LIN {X 0,Y 298.452,Z 269.609,A -85,B 0,C 180,E1 -16435.587,E2 -16435.587} C_VEL
LIN {X 0,Y 298.198,Z 272.62,A -85,B 0,C 180,E1 -16438.768,E2 -16438.768} C_VEL
LIN {X 0,Y 297.924,Z 275.64,A -85,B 0,C 180,E1 -16441.849,E2 -16441.849} C_VEL
LIN {X 0,Y 297.634,Z 279.334,A -85,B 0,C 180,E1 -16445.446,E2 -16445.446} C_VEL
LIN {X 0,Y 302.181,Z 294.942,A -85,B 0,C 180,E1 -16446.632,E2 -16446.632} C_VEL
LIN {X 0,Y 304.72,Z 306.185,A -85,B 0,C 180,E1 -16447.658,E2 -16447.658} C_VEL
LIN {X 0,Y 306.557,Z 317.092,A -85,B 0,C 180,E1 -16448.834,E2 -16448.834} C_VEL
LIN {X 0,Y 305.846,Z 324.673,A -85,B 0,C 180,E1 -16449.662,E2 -16449.662} C_VEL
LIN {X 0,Y 304.462,Z 334.817,A -85,B 0,C 180,E1 -16450.971,E2 -16450.971} C_VEL
LIN {X 0,Y 303.067,Z 344.133,A -85,B 0,C 180,E1 -16452.454,E2 -16452.454} C_VEL
LIN {X 0,Y 301.645,Z 352.621,A -85,B 0,C 180,E1 -16454.112,E2 -16454.112} C_VEL
LIN {X 0,Y 300.146,Z 360.872,A -85,B 0,C 180,E1 -16456.113,E2 -16456.113} C_VEL
LIN {X 0,Y 299.11,Z 366.515,A -85,B 0,C 180,E1 -16457.792,E2 -16457.792} C_VEL
LIN {X 0,Y 298.156,Z 372.013,A -85,B 0,C 180,E1 -16459.817,E2 -16459.817} C_VEL
LIN {X 0,Y 297.455,Z 376.327,A -85,B 0,C 180,E1 -16461.85,E2 -16461.85} C_VEL
LIN {X 0,Y 297.118,Z 378.98,A -85,B 0,C 180,E1 -16463.448,E2 -16463.448} C_VEL
LIN {X 0,Y 296.782,Z 381.858,A -85,B 0,C 180,E1 -16465.926,E2 -16465.926} C_VEL
LIN {X 0,Y 296.535,Z 383.463,A -85,B 0,C 180,E1 -16468.642,E2 -16468.642} C_VEL
LIN {X 0,Y 296.526,Z 383.693,A -85,B 0,C 180,E1 -16470,E2 -16470} C_VEL
LIN {X 0,Y 296.535,Z 383.502,A -85,B 0,C 180,E1 -16471.358,E2 -16471.358} C_VEL
LIN {X 0,Y 296.779,Z 381.947,A -85,B 0,C 180,E1 -16474.074,E2 -16474.074} C_VEL
LIN {X 0,Y 297.086,Z 379.22,A -85,B 0,C 180,E1 -16476.498,E2 -16476.498} C_VEL
LIN {X 0,Y 297.658,Z 375.251,A -85,B 0,C 180,E1 -16478.828,E2 -16478.828} C_VEL
LIN {X 0,Y 298.411,Z 370.618,A -85,B 0,C 180,E1 -16480.86,E2 -16480.86} C_VEL
LIN {X 0,Y 299.685,Z 363.631,A -85,B 0,C 180,E1 -16483.218,E2 -16483.218} C_VEL
LIN {X 0,Y 301.019,Z 356.058,A -85,B 0,C 180,E1 -16485.228,E2 -16485.228} C_VEL
LIN {X 0,Y 302.445,Z 348.294,A -85,B 0,C 180,E1 -16486.886,E2 -16486.886} C_VEL
LIN {X 0,Y 303.98,Z 337.973,A -85,B 0,C 180,E1 -16488.674,E2 -16488.674} C_VEL
LIN {X 0,Y 305.567,Z 326.991,A -85,B 0,C 180,E1 -16490.182,E2 -16490.182} C_VEL
LIN {X 0,Y 306.643,Z 318.121,A -85,B 0,C 180,E1 -16491.16,E2 -16491.16} C_VEL
LIN {X 0,Y 304.903,Z 306.992,A -85,B 0,C 180,E1 -16492.377,E2 -16492.377} C_VEL
LIN {X 0,Y 302.207,Z 294.945,A -85,B 0,C 180,E1 -16493.484,E2 -16493.484} C_VEL
LIN {X 0,Y 298.411,Z 282.147,A -85,B 0,C 180,E1 -16494.464,E2 -16494.464} C_VEL
LIN {X 0,Y 297.654,Z 279.322,A -85,B 0,C 180,E1 -16494.686,E2 -16494.686} C_VEL
LIN {X 0,Y 297.907,Z 275.764,A -85,B 0,C 180,E1 -16498.153,E2 -16498.153} C_VEL
LIN {X 0,Y 298.237,Z 272.051,A -85,B 0,C 180,E1 -16501.967,E2 -16501.967} C_VEL
LIN {X 0,Y 298.43,Z 269.667,A -85,B 0,C 180,E1 -16504.487,E2 -16504.487} C_VEL
LIN {X 0,Y 298.37,Z 266.738,A -85,B 0,C 180,E1 -16507.765,E2 -16507.765} C_VEL
LIN {X 0,Y 298.337,Z 266.319,A -85,B 0,C 180,E1 -16509.498,E2 -16509.498} C_VEL
LIN {X 0,Y 298.372,Z 266.315,A -85,B 0,C 180,E1 -16513.097,E2 -16513.097} C_VEL
LIN {X 0,Y 298.405,Z 266.313,A -85,B 0,C 180,E1 -16516.921,E2 -16516.921} C_VEL
LIN {X 0,Y 298.417,Z 266.311,A -85,B 0,C 180,E1 -16521.004,E2 -16521.004} C_VEL
LIN {X 0,Y 298.423,Z 266.313,A -85,B 0,C 180,E1 -16523.931,E2 -16523.931} C_VEL
LIN {X 0,Y 298.398,Z 266.316,A -85,B 0,C 180,E1 -16527.983,E2 -16527.983} C_VEL
LIN {X 0,Y 298.466,Z 266.307,A -85,B 0,C 180,E1 -16531.904,E2 -16531.904} C_VEL
LIN {X 0,Y 298.487,Z 266.302,A -85,B 0,C 180,E1 -16534.924,E2 -16534.924} C_VEL
LIN {X 0,Y 298.432,Z 266.312,A -85,B 0,C 180,E1 -16539.314,E2 -16539.314} C_VEL
LIN {X 0,Y 298.506,Z 266.299,A -85,B 0,C 180,E1 -16542.177,E2 -16542.177} C_VEL
LIN {X 0,Y 298.56,Z 266.292,A -85,B 0,C 180,E1 -16545.372,E2 -16545.372} C_VEL
LIN {X 0,Y 298.586,Z 266.294,A -85,B 0,C 180,E1 -16549.146,E2 -16549.146} C_VEL
LIN {X 0,Y 298.715,Z 266.277,A -85,B 0,C 180,E1 -16551.239,E2 -16551.239} C_VEL
LIN {X 0,Y 298,Z 266.364,A -85,B 0,C 180,E1 -16552.364,E2 -16552.364} C_VEL
LIN {X 0,Y 295.047,Z 266.73,A -85,B 0,C 180,E1 -16554.192,E2 -16554.192} C_VEL
LIN {X 0,Y 292.654,Z 267.029,A -85,B 0,C 180,E1 -16555.677,E2 -16555.677} C_VEL
LIN {X 0,Y 291.764,Z 267.143,A -85,B 0,C 180,E1 -16556.828,E2 -16556.828} C_VEL
LIN {X 0,Y 291.763,Z 267.142,A -85,B 0,C 180,E1 -16557.217,E2 -16557.217} C_VEL
LIN {X 0,Y 291.862,Z 267.127,A -85,B 0,C 180,E1 -16560,E2 -16560} C_VEL
LIN {X 0,Y 291.79,Z 267.14,A -85,B 0,C 180,E1 -16562.761,E2 -16562.761} C_VEL
LIN {X 0,Y 291.726,Z 267.146,A -85,B 0,C 180,E1 -16566.918,E2 -16566.918} C_VEL
LIN {X 0,Y 291.57,Z 267.164,A -85,B 0,C 180,E1 -16569.714,E2 -16569.714} C_VEL
LIN {X 0,Y 291.524,Z 267.171,A -85,B 0,C 180,E1 -16573.95,E2 -16573.95} C_VEL
LIN {X 0,Y 291.49,Z 267.174,A -85,B 0,C 180,E1 -16576.818,E2 -16576.818} C_VEL
LIN {X 0,Y 291.453,Z 267.181,A -85,B 0,C 180,E1 -16579.875,E2 -16579.875} C_VEL
LIN {X 0,Y 291.349,Z 267.194,A -85,B 0,C 180,E1 -16584.21,E2 -16584.21} C_VEL
LIN {X 0,Y 291.353,Z 267.192,A -85,B 0,C 180,E1 -16587.279,E2 -16587.279} C_VEL
LIN {X 0,Y 291.32,Z 267.196,A -85,B 0,C 180,E1 -16590.439,E2 -16590.439} C_VEL
LIN {X 0,Y 291.346,Z 267.196,A -85,B 0,C 180,E1 -16593.698,E2 -16593.698} C_VEL
LIN {X 0,Y 291.361,Z 267.195,A -85,B 0,C 180,E1 -16597.249,E2 -16597.249} C_VEL
LIN {X 0,Y 291.302,Z 267.2,A -85,B 0,C 180,E1 -16600.648,E2 -16600.648} C_VEL
LIN {X 0,Y 291.373,Z 267.374,A -85,B 0,C 180,E1 -16603.3,E2 -16603.3} C_VEL
LIN {X 0,Y 292.178,Z 271.949,A -85,B 0,C 180,E1 -16607.661,E2 -16607.661} C_VEL
LIN {X 0,Y 292.855,Z 276.179,A -85,B 0,C 180,E1 -16611.394,E2 -16611.394} C_VEL
LIN {X 0,Y 292.993,Z 280.391,A -85,B 0,C 180,E1 -16614.852,E2 -16614.852} C_VEL
LIN {X 0,Y 292.273,Z 284.565,A -85,B 0,C 180,E1 -16618.061,E2 -16618.061} C_VEL
LIN {X 0,Y 291.512,Z 289.748,A -85,B 0,C 180,E1 -16621.958,E2 -16621.958} C_VEL
LIN {X 0,Y 291.018,Z 293.558,A -85,B 0,C 180,E1 -16624.778,E2 -16624.778} C_VEL
LIN {X 0,Y 294.28,Z 306.86,A -85,B 0,C 180,E1 -16625.679,E2 -16625.679} C_VEL
LIN {X 0,Y 296.52,Z 318.834,A -85,B 0,C 180,E1 -16626.69,E2 -16626.69} C_VEL
LIN {X 0,Y 297.9,Z 330.098,A -85,B 0,C 180,E1 -16627.823,E2 -16627.823} C_VEL
LIN {X 0,Y 298.47,Z 339.723,A -85,B 0,C 180,E1 -16628.956,E2 -16628.956} C_VEL
LIN {X 0,Y 296.712,Z 351.254,A -85,B 0,C 180,E1 -16630.454,E2 -16630.454} C_VEL
LIN {X 0,Y 295.154,Z 360.542,A -85,B 0,C 180,E1 -16631.968,E2 -16631.968} C_VEL
LIN {X 0,Y 293.746,Z 369.016,A -85,B 0,C 180,E1 -16633.673,E2 -16633.673} C_VEL
LIN {X 0,Y 292.32,Z 377.289,A -85,B 0,C 180,E1 -16635.733,E2 -16635.733} C_VEL
LIN {X 0,Y 291.092,Z 383.957,A -85,B 0,C 180,E1 -16637.804,E2 -16637.804} C_VEL
LIN {X 0,Y 290.208,Z 390.063,A -85,B 0,C 180,E1 -16640.24,E2 -16640.24} C_VEL
LIN {X 0,Y 289.72,Z 394.033,A -85,B 0,C 180,E1 -16642.333,E2 -16642.333} C_VEL
LIN {X 0,Y 289.475,Z 397.064,A -85,B 0,C 180,E1 -16644.513,E2 -16644.513} C_VEL
LIN {X 0,Y 289.438,Z 399.365,A -85,B 0,C 180,E1 -16647.216,E2 -16647.216} C_VEL
LIN {X 0,Y 289.415,Z 399.972,A -85,B 0,C 180,E1 -16648.608,E2 -16648.608} C_VEL
LIN {X 0,Y 289.437,Z 400.186,A -85,B 0,C 180,E1 -16650,E2 -16650} C_VEL
LIN {X 0,Y 289.414,Z 399.965,A -85,B 0,C 180,E1 -16651.391,E2 -16651.391} C_VEL
LIN {X 0,Y 289.434,Z 399.353,A -85,B 0,C 180,E1 -16652.783,E2 -16652.783} C_VEL
LIN {X 0,Y 289.429,Z 397.143,A -85,B 0,C 180,E1 -16655.391,E2 -16655.391} C_VEL
LIN {X 0,Y 289.719,Z 393.998,A -85,B 0,C 180,E1 -16657.667,E2 -16657.667} C_VEL
LIN {X 0,Y 290.208,Z 390.012,A -85,B 0,C 180,E1 -16659.76,E2 -16659.76} C_VEL
LIN {X 0,Y 291.091,Z 383.887,A -85,B 0,C 180,E1 -16662.196,E2 -16662.196} C_VEL
LIN {X 0,Y 292.303,Z 377.203,A -85,B 0,C 180,E1 -16664.267,E2 -16664.267} C_VEL
LIN {X 0,Y 293.791,Z 368.912,A -85,B 0,C 180,E1 -16666.325,E2 -16666.325} C_VEL
LIN {X 0,Y 295.165,Z 360.409,A -85,B 0,C 180,E1 -16668.031,E2 -16668.031} C_VEL
LIN {X 0,Y 296.87,Z 349.907,A -85,B 0,C 180,E1 -16669.715,E2 -16669.715} C_VEL
LIN {X 0,Y 298.404,Z 339.517,A -85,B 0,C 180,E1 -16671.049,E2 -16671.049} C_VEL
LIN {X 0,Y 297.673,Z 328.312,A -85,B 0,C 180,E1 -16672.351,E2 -16672.351} C_VEL
LIN {X 0,Y 296.062,Z 316.214,A -85,B 0,C 180,E1 -16673.524,E2 -16673.524} C_VEL
LIN {X 0,Y 293.553,Z 303.653,A -85,B 0,C 180,E1 -16674.527,E2 -16674.527} C_VEL
LIN {X 0,Y 291.013,Z 293.527,A -85,B 0,C 180,E1 -16675.21,E2 -16675.21} C_VEL
LIN {X 0,Y 291.631,Z 288.68,A -85,B 0,C 180,E1 -16678.815,E2 -16678.815} C_VEL
LIN {X 0,Y 292.447,Z 283.451,A -85,B 0,C 180,E1 -16682.742,E2 -16682.742} C_VEL
LIN {X 0,Y 292.978,Z 280.087,A -85,B 0,C 180,E1 -16685.353,E2 -16685.353} C_VEL
LIN {X 0,Y 292.849,Z 276.136,A -85,B 0,C 180,E1 -16688.606,E2 -16688.606} C_VEL
LIN {X 0,Y 292.145,Z 271.902,A -85,B 0,C 180,E1 -16692.344,E2 -16692.344} C_VEL
LIN {X 0,Y 291.365,Z 267.243,A -85,B 0,C 180,E1 -16696.779,E2 -16696.779} C_VEL
LIN {X 0,Y 291.335,Z 267.196,A -85,B 0,C 180,E1 -16701.155,E2 -16701.155} C_VEL
LIN {X 0,Y 291.356,Z 267.195,A -85,B 0,C 180,E1 -16704.625,E2 -16704.625} C_VEL
LIN {X 0,Y 291.367,Z 267.194,A -85,B 0,C 180,E1 -16707.95,E2 -16707.95} C_VEL
LIN {X 0,Y 291.344,Z 267.194,A -85,B 0,C 180,E1 -16711.154,E2 -16711.154} C_VEL
LIN {X 0,Y 291.349,Z 267.196,A -85,B 0,C 180,E1 -16714.266,E2 -16714.266} C_VEL
LIN {X 0,Y 291.362,Z 267.191,A -85,B 0,C 180,E1 -16717.298,E2 -16717.298} C_VEL
LIN {X 0,Y 291.459,Z 267.18,A -85,B 0,C 180,E1 -16720.27,E2 -16720.27} C_VEL
LIN {X 0,Y 291.556,Z 267.165,A -85,B 0,C 180,E1 -16724.624,E2 -16724.624} C_VEL
LIN {X 0,Y 291.53,Z 267.169,A -85,B 0,C 180,E1 -16728.88,E2 -16728.88} C_VEL
LIN {X 0,Y 291.669,Z 267.154,A -85,B 0,C 180,E1 -16731.687,E2 -16731.687} C_VEL
LIN {X 0,Y 291.625,Z 267.156,A -85,B 0,C 180,E1 -16734.468,E2 -16734.468} C_VEL
LIN {X 0,Y 291.89,Z 267.123,A -85,B 0,C 180,E1 -16738.62,E2 -16738.62} C_VEL
LIN {X 0,Y 291.881,Z 267.127,A -85,B 0,C 180,E1 -16741.38,E2 -16741.38} C_VEL
LIN {X 0,Y 291.714,Z 267.15,A -85,B 0,C 180,E1 -16746.919,E2 -16746.919} C_VEL
LIN {X 0,Y 291.569,Z 267.164,A -85,B 0,C 180,E1 -16749.714,E2 -16749.714} C_VEL
LIN {X 0,Y 291.517,Z 267.17,A -85,B 0,C 180,E1 -16753.951,E2 -16753.951} C_VEL
LIN {X 0,Y 291.44,Z 267.182,A -85,B 0,C 180,E1 -16758.27,E2 -16758.27} C_VEL
LIN {X 0,Y 291.36,Z 267.189,A -85,B 0,C 180,E1 -16761.212,E2 -16761.212} C_VEL
LIN {X 0,Y 291.385,Z 267.19,A -85,B 0,C 180,E1 -16764.207,E2 -16764.207} C_VEL
LIN {X 0,Y 291.426,Z 267.181,A -85,B 0,C 180,E1 -16767.271,E2 -16767.271} C_VEL
LIN {X 0,Y 291.34,Z 267.195,A -85,B 0,C 180,E1 -16770.437,E2 -16770.437} C_VEL
LIN {X 0,Y 291.346,Z 267.194,A -85,B 0,C 180,E1 -16773.698,E2 -16773.698} C_VEL
LIN {X 0,Y 291.381,Z 267.188,A -85,B 0,C 180,E1 -16777.255,E2 -16777.255} C_VEL
LIN {X 0,Y 291.335,Z 267.194,A -85,B 0,C 180,E1 -16780.643,E2 -16780.643} C_VEL
LIN {X 0,Y 291.291,Z 267.199,A -85,B 0,C 180,E1 -16784.402,E2 -16784.402} C_VEL
LIN {X 0,Y 291.295,Z 267.2,A -85,B 0,C 180,E1 -16788.412,E2 -16788.412} C_VEL
LIN {X 0,Y 291.294,Z 267.202,A -85,B 0,C 180,E1 -16791.149,E2 -16791.149} C_VEL
LIN {X 0,Y 291.405,Z 268.296,A -85,B 0,C 180,E1 -16792.919,E2 -16792.919} C_VEL
LIN {X 0,Y 291.36,Z 271.305,A -85,B 0,C 180,E1 -16796.304,E2 -16796.304} C_VEL
LIN {X 0,Y 291.043,Z 275.128,A -85,B 0,C 180,E1 -16800.38,E2 -16800.38} C_VEL
LIN {X 0,Y 290.656,Z 279.54,A -85,B 0,C 180,E1 -16804.816,E2 -16804.816} C_VEL
LIN {X 0,Y 295.227,Z 295.045,A -85,B 0,C 180,E1 -16806.04,E2 -16806.04} C_VEL
LIN {X 0,Y 297.691,Z 305.584,A -85,B 0,C 180,E1 -16807.033,E2 -16807.033} C_VEL
LIN {X 0,Y 299.638,Z 317.307,A -85,B 0,C 180,E1 -16808.321,E2 -16808.321} C_VEL
LIN {X 0,Y 299.789,Z 320.451,A -85,B 0,C 180,E1 -16808.693,E2 -16808.693} C_VEL
LIN {X 0,Y 298.258,Z 331.498,A -85,B 0,C 180,E1 -16810.021,E2 -16810.021} C_VEL
LIN {X 0,Y 296.763,Z 341.17,A -85,B 0,C 180,E1 -16811.487,E2 -16811.487} C_VEL
LIN {X 0,Y 295.115,Z 351.228,A -85,B 0,C 180,E1 -16813.395,E2 -16813.395} C_VEL
LIN {X 0,Y 293.459,Z 359.848,A -85,B 0,C 180,E1 -16815.436,E2 -16815.436} C_VEL
LIN {X 0,Y 292.168,Z 366.716,A -85,B 0,C 180,E1 -16817.497,E2 -16817.497} C_VEL
LIN {X 0,Y 291.165,Z 372.214,A -85,B 0,C 180,E1 -16819.57,E2 -16819.57} C_VEL
LIN {X 0,Y 290.436,Z 376.528,A -85,B 0,C 180,E1 -16821.652,E2 -16821.652} C_VEL
LIN {X 0,Y 290.034,Z 379.43,A -85,B 0,C 180,E1 -16823.464,E2 -16823.464} C_VEL
LIN {X 0,Y 289.704,Z 382.058,A -85,B 0,C 180,E1 -16825.827,E2 -16825.827} C_VEL
LIN {X 0,Y 289.456,Z 383.662,A -85,B 0,C 180,E1 -16828.609,E2 -16828.609} C_VEL
LIN {X 0,Y 289.443,Z 383.893,A -85,B 0,C 180,E1 -16830,E2 -16830} C_VEL
LIN {X 0,Y 289.456,Z 383.701,A -85,B 0,C 180,E1 -16831.391,E2 -16831.391} C_VEL
LIN {X 0,Y 289.558,Z 383.114,A -85,B 0,C 180,E1 -16832.783,E2 -16832.783} C_VEL
LIN {X 0,Y 289.701,Z 382.146,A -85,B 0,C 180,E1 -16834.174,E2 -16834.174} C_VEL
LIN {X 0,Y 290.011,Z 379.625,A -85,B 0,C 180,E1 -16836.495,E2 -16836.495} C_VEL
LIN {X 0,Y 290.468,Z 376.728,A -85,B 0,C 180,E1 -16838.347,E2 -16838.347} C_VEL
LIN {X 0,Y 291.138,Z 372.478,A -85,B 0,C 180,E1 -16840.431,E2 -16840.431} C_VEL
LIN {X 0,Y 292.325,Z 366.037,A -85,B 0,C 180,E1 -16842.849,E2 -16842.849} C_VEL
LIN {X 0,Y 293.647,Z 358.958,A -85,B 0,C 180,E1 -16844.909,E2 -16844.909} C_VEL
LIN {X 0,Y 295.346,Z 350.134,A -85,B 0,C 180,E1 -16846.948,E2 -16846.948} C_VEL
LIN {X 0,Y 296.819,Z 341.07,A -85,B 0,C 180,E1 -16848.644,E2 -16848.644} C_VEL
LIN {X 0,Y 298.311,Z 331.053,A -85,B 0,C 180,E1 -16850.155,E2 -16850.155} C_VEL
LIN {X 0,Y 299.884,Z 319.891,A -85,B 0,C 180,E1 -16851.481,E2 -16851.481} C_VEL
LIN {X 0,Y 298.563,Z 310.14,A -85,B 0,C 180,E1 -16852.606,E2 -16852.606} C_VEL
LIN {X 0,Y 296.022,Z 298.109,A -85,B 0,C 180,E1 -16853.804,E2 -16853.804} C_VEL
LIN {X 0,Y 292.397,Z 285.232,A -85,B 0,C 180,E1 -16854.88,E2 -16854.88} C_VEL
LIN {X 0,Y 290.638,Z 279.573,A -85,B 0,C 180,E1 -16855.277,E2 -16855.277} C_VEL
LIN {X 0,Y 290.944,Z 275.962,A -85,B 0,C 180,E1 -16858.889,E2 -16858.889} C_VEL
LIN {X 0,Y 291.236,Z 272.66,A -85,B 0,C 180,E1 -16862.37,E2 -16862.37} C_VEL
LIN {X 0,Y 291.395,Z 269.922,A -85,B 0,C 180,E1 -16865.369,E2 -16865.369} C_VEL
LIN {X 0,Y 291.386,Z 268.263,A -85,B 0,C 180,E1 -16867.256,E2 -16867.256} C_VEL
LIN {X 0,Y 291.29,Z 267.199,A -85,B 0,C 180,E1 -16868.852,E2 -16868.852} C_VEL
LIN {X 0,Y 291.288,Z 267.199,A -85,B 0,C 180,E1 -16872.498,E2 -16872.498} C_VEL
LIN {X 0,Y 291.312,Z 267.199,A -85,B 0,C 180,E1 -16876.366,E2 -16876.366} C_VEL
LIN {X 0,Y 291.389,Z 267.188,A -85,B 0,C 180,E1 -16880.517,E2 -16880.517} C_VEL
LIN {X 0,Y 291.416,Z 267.182,A -85,B 0,C 180,E1 -16882.921,E2 -16882.921} C_VEL
LIN {X 0,Y 291.347,Z 267.194,A -85,B 0,C 180,E1 -16886.302,E2 -16886.302} C_VEL
LIN {X 0,Y 291.39,Z 267.188,A -85,B 0,C 180,E1 -16890.26,E2 -16890.26} C_VEL
LIN {X 0,Y 291.419,Z 267.184,A -85,B 0,C 180,E1 -16894.272,E2 -16894.272} C_VEL
LIN {X 0,Y 291.375,Z 267.188,A -85,B 0,C 180,E1 -16897.299,E2 -16897.299} C_VEL
LIN {X 0,Y 291.442,Z 267.179,A -85,B 0,C 180,E1 -16900.269,E2 -16900.269} C_VEL
LIN {X 0,Y 291.5,Z 267.173,A -85,B 0,C 180,E1 -16904.665,E2 -16904.665} C_VEL
LIN {X 0,Y 291.532,Z 267.17,A -85,B 0,C 180,E1 -16908.88,E2 -16908.88} C_VEL
LIN {X 0,Y 291.667,Z 267.152,A -85,B 0,C 180,E1 -16911.687,E2 -16911.687} C_VEL
LIN {X 0,Y 291.609,Z 267.159,A -85,B 0,C 180,E1 -16914.468,E2 -16914.468} C_VEL
LIN {X 0,Y 291.763,Z 267.142,A -85,B 0,C 180,E1 -16917.217,E2 -16917.217} C_VEL
LIN {X 0,Y 291.303,Z 267.207,A -85,B 0,C 180,E1 -16918.37,E2 -16918.37} C_VEL
LIN {X 0,Y 289.813,Z 267.396,A -85,B 0,C 180,E1 -16919.503,E2 -16919.503} C_VEL
LIN {X 0,Y 285.995,Z 267.866,A -85,B 0,C 180,E1 -16921.773,E2 -16921.773} C_VEL
LIN {X 0,Y 284.788,Z 268.011,A -85,B 0,C 180,E1 -16922.954,E2 -16922.954} C_VEL
LIN {X 0,Y 284.636,Z 268.028,A -85,B 0,C 180,E1 -16923.356,E2 -16923.356} C_VEL
LIN {X 0,Y 284.676,Z 268.023,A -85,B 0,C 180,E1 -16927.091,E2 -16927.091} C_VEL
LIN {X 0,Y 284.516,Z 268.044,A -85,B 0,C 180,E1 -16929.957,E2 -16929.957} C_VEL
LIN {X 0,Y 284.484,Z 268.05,A -85,B 0,C 180,E1 -16934.303,E2 -16934.303} C_VEL
LIN {X 0,Y 284.428,Z 268.053,A -85,B 0,C 180,E1 -16937.248,E2 -16937.248} C_VEL
LIN {X 0,Y 284.379,Z 268.063,A -85,B 0,C 180,E1 -16940.242,E2 -16940.242} C_VEL
LIN {X 0,Y 284.313,Z 268.071,A -85,B 0,C 180,E1 -16943.849,E2 -16943.849} C_VEL
LIN {X 0,Y 284.283,Z 268.075,A -85,B 0,C 180,E1 -16948.016,E2 -16948.016} C_VEL
LIN {X 0,Y 284.287,Z 268.073,A -85,B 0,C 180,E1 -16951.275,E2 -16951.275} C_VEL
LIN {X 0,Y 284.338,Z 268.069,A -85,B 0,C 180,E1 -16955.347,E2 -16955.347} C_VEL
LIN {X 0,Y 284.299,Z 268.072,A -85,B 0,C 180,E1 -16958.171,E2 -16958.171} C_VEL
LIN {X 0,Y 284.27,Z 268.074,A -85,B 0,C 180,E1 -16962.445,E2 -16962.445} C_VEL
LIN {X 0,Y 284.831,Z 271.136,A -85,B 0,C 180,E1 -16965.689,E2 -16965.689} C_VEL
LIN {X 0,Y 285.565,Z 275.42,A -85,B 0,C 180,E1 -16969.724,E2 -16969.724} C_VEL
LIN {X 0,Y 285.969,Z 279.157,A -85,B 0,C 180,E1 -16972.978,E2 -16972.978} C_VEL
LIN {X 0,Y 285.796,Z 282.295,A -85,B 0,C 180,E1 -16975.556,E2 -16975.556} C_VEL
LIN {X 0,Y 284.876,Z 287.6,A -85,B 0,C 180,E1 -16979.708,E2 -16979.708} C_VEL
LIN {X 0,Y 284.072,Z 293.09,A -85,B 0,C 180,E1 -16983.916,E2 -16983.916} C_VEL
LIN {X 0,Y 284.061,Z 293.365,A -85,B 0,C 180,E1 -16984.115,E2 -16984.115} C_VEL
LIN {X 0,Y 287.328,Z 306.368,A -85,B 0,C 180,E1 -16985.032,E2 -16985.032} C_VEL
LIN {X 0,Y 289.612,Z 318.46,A -85,B 0,C 180,E1 -16986.085,E2 -16986.085} C_VEL
LIN {X 0,Y 291.063,Z 329.895,A -85,B 0,C 180,E1 -16987.273,E2 -16987.273} C_VEL
LIN {X 0,Y 291.653,Z 340.956,A -85,B 0,C 180,E1 -16988.625,E2 -16988.625} C_VEL
LIN {X 0,Y 289.82,Z 352.186,A -85,B 0,C 180,E1 -16990.154,E2 -16990.154} C_VEL
LIN {X 0,Y 288.038,Z 362.07,A -85,B 0,C 180,E1 -16991.86,E2 -16991.86} C_VEL
LIN {X 0,Y 286.628,Z 370.309,A -85,B 0,C 180,E1 -16993.622,E2 -16993.622} C_VEL
LIN {X 0,Y 285.177,Z 378.327,A -85,B 0,C 180,E1 -16995.733,E2 -16995.733} C_VEL
LIN {X 0,Y 283.985,Z 384.754,A -85,B 0,C 180,E1 -16997.857,E2 -16997.857} C_VEL
LIN {X 0,Y 283.183,Z 389.863,A -85,B 0,C 180,E1 -16999.995,E2 -16999.995} C_VEL
LIN {X 0,Y 282.676,Z 393.834,A -85,B 0,C 180,E1 -17002.14,E2 -17002.14} C_VEL
LIN {X 0,Y 282.37,Z 397.103,A -85,B 0,C 180,E1 -17004.609,E2 -17004.609} C_VEL
LIN {X 0,Y 282.346,Z 399.165,A -85,B 0,C 180,E1 -17007.146,E2 -17007.146} C_VEL
LIN {X 0,Y 282.338,Z 399.773,A -85,B 0,C 180,E1 -17008.573,E2 -17008.573} C_VEL
LIN {X 0,Y 282.356,Z 399.987,A -85,B 0,C 180,E1 -17010,E2 -17010} C_VEL
LIN {X 0,Y 282.337,Z 399.765,A -85,B 0,C 180,E1 -17011.426,E2 -17011.426} C_VEL
LIN {X 0,Y 282.341,Z 399.153,A -85,B 0,C 180,E1 -17012.853,E2 -17012.853} C_VEL
LIN {X 0,Y 282.34,Z 397.148,A -85,B 0,C 180,E1 -17015.326,E2 -17015.326} C_VEL
LIN {X 0,Y 282.675,Z 393.797,A -85,B 0,C 180,E1 -17017.859,E2 -17017.859} C_VEL
LIN {X 0,Y 283.183,Z 389.811,A -85,B 0,C 180,E1 -17020.004,E2 -17020.004} C_VEL
LIN {X 0,Y 284.118,Z 383.684,A -85,B 0,C 180,E1 -17022.5,E2 -17022.5} C_VEL
LIN {X 0,Y 285.411,Z 377.001,A -85,B 0,C 180,E1 -17024.619,E2 -17024.619} C_VEL
LIN {X 0,Y 286.966,Z 368.71,A -85,B 0,C 180,E1 -17026.724,E2 -17026.724} C_VEL
LIN {X 0,Y 288.381,Z 360.205,A -85,B 0,C 180,E1 -17028.47,E2 -17028.47} C_VEL
LIN {X 0,Y 290.181,Z 349.703,A -85,B 0,C 180,E1 -17030.189,E2 -17030.189} C_VEL
LIN {X 0,Y 291.603,Z 340.743,A -85,B 0,C 180,E1 -17031.379,E2 -17031.379} C_VEL
LIN {X 0,Y 291.158,Z 331.405,A -85,B 0,C 180,E1 -17032.532,E2 -17032.532} C_VEL
LIN {X 0,Y 289.588,Z 318.372,A -85,B 0,C 180,E1 -17033.893,E2 -17033.893} C_VEL
LIN {X 0,Y 287.147,Z 305.668,A -85,B 0,C 180,E1 -17034.994,E2 -17034.994} C_VEL
LIN {X 0,Y 284.062,Z 293.324,A -85,B 0,C 180,E1 -17035.875,E2 -17035.875} C_VEL
LIN {X 0,Y 284.725,Z 288.481,A -85,B 0,C 180,E1 -17039.582,E2 -17039.582} C_VEL
LIN {X 0,Y 285.526,Z 283.824,A -85,B 0,C 180,E1 -17043.187,E2 -17043.187} C_VEL
LIN {X 0,Y 285.941,Z 280.155,A -85,B 0,C 180,E1 -17046.149,E2 -17046.149} C_VEL
LIN {X 0,Y 285.869,Z 277.83,A -85,B 0,C 180,E1 -17048.121,E2 -17048.121} C_VEL
LIN {X 0,Y 285.552,Z 275.379,A -85,B 0,C 180,E1 -17050.273,E2 -17050.273} C_VEL
LIN {X 0,Y 284.825,Z 271.089,A -85,B 0,C 180,E1 -17054.31,E2 -17054.31} C_VEL
LIN {X 0,Y 284.256,Z 268.074,A -85,B 0,C 180,E1 -17057.328,E2 -17057.328} C_VEL
LIN {X 0,Y 284.283,Z 268.077,A -85,B 0,C 180,E1 -17060.03,E2 -17060.03} C_VEL
LIN {X 0,Y 284.322,Z 268.068,A -85,B 0,C 180,E1 -17063.612,E2 -17063.612} C_VEL
LIN {X 0,Y 284.307,Z 268.072,A -85,B 0,C 180,E1 -17067.19,E2 -17067.19} C_VEL
LIN {X 0,Y 284.338,Z 268.071,A -85,B 0,C 180,E1 -17070.374,E2 -17070.374} C_VEL
LIN {X 0,Y 284.3,Z 268.073,A -85,B 0,C 180,E1 -17073.579,E2 -17073.579} C_VEL
LIN {X 0,Y 284.321,Z 268.069,A -85,B 0,C 180,E1 -17076.703,E2 -17076.703} C_VEL
LIN {X 0,Y 284.388,Z 268.062,A -85,B 0,C 180,E1 -17079.898,E2 -17079.898} C_VEL
LIN {X 0,Y 284.493,Z 268.046,A -85,B 0,C 180,E1 -17084.459,E2 -17084.459} C_VEL
LIN {X 0,Y 284.484,Z 268.046,A -85,B 0,C 180,E1 -17088.601,E2 -17088.601} C_VEL
LIN {X 0,Y 284.623,Z 268.033,A -85,B 0,C 180,E1 -17091.48,E2 -17091.48} C_VEL
LIN {X 0,Y 284.594,Z 268.032,A -85,B 0,C 180,E1 -17094.331,E2 -17094.331} C_VEL
LIN {X 0,Y 284.856,Z 267.999,A -85,B 0,C 180,E1 -17098.586,E2 -17098.586} C_VEL
LIN {X 0,Y 284.848,Z 268.003,A -85,B 0,C 180,E1 -17101.414,E2 -17101.414} C_VEL
LIN {X 0,Y 284.667,Z 268.027,A -85,B 0,C 180,E1 -17107.091,E2 -17107.091} C_VEL
LIN {X 0,Y 284.515,Z 268.042,A -85,B 0,C 180,E1 -17109.957,E2 -17109.957} C_VEL
LIN {X 0,Y 284.465,Z 268.05,A -85,B 0,C 180,E1 -17114.304,E2 -17114.304} C_VEL
LIN {X 0,Y 284.376,Z 268.063,A -85,B 0,C 180,E1 -17118.74,E2 -17118.74} C_VEL
LIN {X 0,Y 284.316,Z 268.067,A -85,B 0,C 180,E1 -17121.764,E2 -17121.764} C_VEL
LIN {X 0,Y 284.34,Z 268.066,A -85,B 0,C 180,E1 -17124.847,E2 -17124.847} C_VEL
LIN {X 0,Y 284.365,Z 268.064,A -85,B 0,C 180,E1 -17128.007,E2 -17128.007} C_VEL
LIN {X 0,Y 284.298,Z 268.069,A -85,B 0,C 180,E1 -17131.274,E2 -17131.274} C_VEL
LIN {X 0,Y 284.342,Z 268.065,A -85,B 0,C 180,E1 -17135.348,E2 -17135.348} C_VEL
LIN {X 0,Y 284.319,Z 268.07,A -85,B 0,C 180,E1 -17138.168,E2 -17138.168} C_VEL
LIN {X 0,Y 284.27,Z 268.074,A -85,B 0,C 180,E1 -17142.124,E2 -17142.124} C_VEL
LIN {X 0,Y 284.238,Z 268.079,A -85,B 0,C 180,E1 -17146.186,E2 -17146.186} C_VEL
LIN {X 0,Y 284.255,Z 268.078,A -85,B 0,C 180,E1 -17150.037,E2 -17150.037} C_VEL
LIN {X 0,Y 284.29,Z 268.487,A -85,B 0,C 180,E1 -17151.828,E2 -17151.828} C_VEL
LIN {X 0,Y 284.362,Z 271.498,A -85,B 0,C 180,E1 -17155.358,E2 -17155.358} C_VEL
LIN {X 0,Y 284.114,Z 274.518,A -85,B 0,C 180,E1 -17158.703,E2 -17158.703} C_VEL
LIN {X 0,Y 283.815,Z 277.587,A -85,B 0,C 180,E1 -17161.934,E2 -17161.934} C_VEL
LIN {X 0,Y 283.678,Z 279.774,A -85,B 0,C 180,E1 -17164.175,E2 -17164.175} C_VEL
LIN {X 0,Y 287.811,Z 293.52,A -85,B 0,C 180,E1 -17165.27,E2 -17165.27} C_VEL
LIN {X 0,Y 290.503,Z 304.226,A -85,B 0,C 180,E1 -17166.298,E2 -17166.298} C_VEL
LIN {X 0,Y 292.587,Z 315.797,A -85,B 0,C 180,E1 -17167.585,E2 -17167.585} C_VEL
LIN {X 0,Y 293.16,Z 320.657,A -85,B 0,C 180,E1 -17168.187,E2 -17168.187} C_VEL
LIN {X 0,Y 291.589,Z 331.702,A -85,B 0,C 180,E1 -17169.544,E2 -17169.544} C_VEL
LIN {X 0,Y 289.929,Z 341.982,A -85,B 0,C 180,E1 -17171.149,E2 -17171.149} C_VEL
LIN {X 0,Y 288.319,Z 351.43,A -85,B 0,C 180,E1 -17172.992,E2 -17172.992} C_VEL
LIN {X 0,Y 286.602,Z 360.049,A -85,B 0,C 180,E1 -17175.08,E2 -17175.08} C_VEL
LIN {X 0,Y 285.237,Z 366.918,A -85,B 0,C 180,E1 -17177.188,E2 -17177.188} C_VEL
LIN {X 0,Y 284.189,Z 372.415,A -85,B 0,C 180,E1 -17179.311,E2 -17179.311} C_VEL
LIN {X 0,Y 283.405,Z 376.729,A -85,B 0,C 180,E1 -17181.443,E2 -17181.443} C_VEL
LIN {X 0,Y 282.922,Z 379.918,A -85,B 0,C 180,E1 -17183.532,E2 -17183.532} C_VEL
LIN {X 0,Y 282.628,Z 382.258,A -85,B 0,C 180,E1 -17185.722,E2 -17185.722} C_VEL
LIN {X 0,Y 282.491,Z 383.25,A -85,B 0,C 180,E1 -17187.148,E2 -17187.148} C_VEL
LIN {X 0,Y 282.363,Z 384.092,A -85,B 0,C 180,E1 -17190,E2 -17190} C_VEL
LIN {X 0,Y 282.38,Z 383.9,A -85,B 0,C 180,E1 -17191.426,E2 -17191.426} C_VEL
LIN {X 0,Y 282.49,Z 383.313,A -85,B 0,C 180,E1 -17192.852,E2 -17192.852} C_VEL
LIN {X 0,Y 282.625,Z 382.346,A -85,B 0,C 180,E1 -17194.278,E2 -17194.278} C_VEL
LIN {X 0,Y 282.943,Z 380.013,A -85,B 0,C 180,E1 -17196.505,E2 -17196.505} C_VEL
LIN {X 0,Y 283.424,Z 376.928,A -85,B 0,C 180,E1 -17198.556,E2 -17198.556} C_VEL
LIN {X 0,Y 284.164,Z 372.676,A -85,B 0,C 180,E1 -17200.69,E2 -17200.69} C_VEL
LIN {X 0,Y 285.415,Z 366.235,A -85,B 0,C 180,E1 -17203.166,E2 -17203.166} C_VEL
LIN {X 0,Y 286.774,Z 359.156,A -85,B 0,C 180,E1 -17205.275,E2 -17205.275} C_VEL
LIN {X 0,Y 288.575,Z 350.331,A -85,B 0,C 180,E1 -17207.358,E2 -17207.358} C_VEL
LIN {X 0,Y 290.163,Z 340.897,A -85,B 0,C 180,E1 -17209.158,E2 -17209.158} C_VEL
LIN {X 0,Y 291.874,Z 329.959,A -85,B 0,C 180,E1 -17210.804,E2 -17210.804} C_VEL
LIN {X 0,Y 293.141,Z 320.09,A -85,B 0,C 180,E1 -17212,E2 -17212} C_VEL
LIN {X 0,Y 291.46,Z 308.967,A -85,B 0,C 180,E1 -17213.32,E2 -17213.32} C_VEL
LIN {X 0,Y 288.82,Z 297.087,A -85,B 0,C 180,E1 -17214.527,E2 -17214.527} C_VEL
LIN {X 0,Y 285.113,Z 284.593,A -85,B 0,C 180,E1 -17215.597,E2 -17215.597} C_VEL
LIN {X 0,Y 283.691,Z 279.759,A -85,B 0,C 180,E1 -17215.964,E2 -17215.964} C_VEL
LIN {X 0,Y 284.017,Z 275.853,A -85,B 0,C 180,E1 -17219.994,E2 -17219.994} C_VEL
LIN {X 0,Y 284.228,Z 273.141,A -85,B 0,C 180,E1 -17222.956,E2 -17222.956} C_VEL
LIN {X 0,Y 284.345,Z 270.116,A -85,B 0,C 180,E1 -17226.384,E2 -17226.384} C_VEL
LIN {X 0,Y 284.285,Z 268.601,A -85,B 0,C 180,E1 -17228.174,E2 -17228.174} C_VEL
LIN {X 0,Y 284.254,Z 268.074,A -85,B 0,C 180,E1 -17230.004,E2 -17230.004} C_VEL
LIN {X 0,Y 284.236,Z 268.078,A -85,B 0,C 180,E1 -17234.188,E2 -17234.188} C_VEL
LIN {X 0,Y 284.274,Z 268.076,A -85,B 0,C 180,E1 -17238.124,E2 -17238.124} C_VEL
LIN {X 0,Y 284.331,Z 268.069,A -85,B 0,C 180,E1 -17242.276,E2 -17242.276} C_VEL
LIN {X 0,Y 284.311,Z 268.069,A -85,B 0,C 180,E1 -17245.351,E2 -17245.351} C_VEL
LIN {X 0,Y 284.298,Z 268.068,A -85,B 0,C 180,E1 -17248.726,E2 -17248.726} C_VEL
LIN {X 0,Y 284.4,Z 268.055,A -85,B 0,C 180,E1 -17252.826,E2 -17252.826} C_VEL
LIN {X 0,Y 284.335,Z 268.062,A -85,B 0,C 180,E1 -17256.704,E2 -17256.704} C_VEL
LIN {X 0,Y 284.379,Z 268.061,A -85,B 0,C 180,E1 -17259.904,E2 -17259.904} C_VEL
LIN {X 0,Y 284.45,Z 268.051,A -85,B 0,C 180,E1 -17264.492,E2 -17264.492} C_VEL
LIN {X 0,Y 284.485,Z 268.046,A -85,B 0,C 180,E1 -17268.601,E2 -17268.601} C_VEL
LIN {X 0,Y 284.622,Z 268.031,A -85,B 0,C 180,E1 -17271.48,E2 -17271.48} C_VEL
LIN {X 0,Y 284.579,Z 268.034,A -85,B 0,C 180,E1 -17274.331,E2 -17274.331} C_VEL
LIN {X 0,Y 284.842,Z 268.005,A -85,B 0,C 180,E1 -17278.586,E2 -17278.586} C_VEL
LIN {X 0,Y 284.856,Z 268,A -85,B 0,C 180,E1 -17281.414,E2 -17281.414} C_VEL
LIN {X 0,Y 284.636,Z 268.028,A -85,B 0,C 180,E1 -17283.356,E2 -17283.356} C_VEL
LIN {X 0,Y 283.843,Z 268.13,A -85,B 0,C 180,E1 -17284.537,E2 -17284.537} C_VEL
LIN {X 0,Y 281.005,Z 268.484,A -85,B 0,C 180,E1 -17286.464,E2 -17286.464} C_VEL
LIN {X 0,Y 278.652,Z 268.774,A -85,B 0,C 180,E1 -17288.029,E2 -17288.029} C_VEL
LIN {X 0,Y 277.607,Z 268.904,A -85,B 0,C 180,E1 -17289.239,E2 -17289.239} C_VEL
LIN {X 0,Y 277.496,Z 268.917,A -85,B 0,C 180,E1 -17289.648,E2 -17289.648} C_VEL
LIN {X 0,Y 277.417,Z 268.927,A -85,B 0,C 180,E1 -17293.18,E2 -17293.18} C_VEL
LIN {X 0,Y 277.409,Z 268.932,A -85,B 0,C 180,E1 -17296.181,E2 -17296.181} C_VEL
LIN {X 0,Y 277.346,Z 268.938,A -85,B 0,C 180,E1 -17300.349,E2 -17300.349} C_VEL
LIN {X 0,Y 277.254,Z 268.95,A -85,B 0,C 180,E1 -17304.139,E2 -17304.139} C_VEL
LIN {X 0,Y 277.269,Z 268.947,A -85,B 0,C 180,E1 -17307.482,E2 -17307.482} C_VEL
LIN {X 0,Y 277.249,Z 268.949,A -85,B 0,C 180,E1 -17310.473,E2 -17310.473} C_VEL
LIN {X 0,Y 277.247,Z 268.953,A -85,B 0,C 180,E1 -17313.896,E2 -17313.896} C_VEL
LIN {X 0,Y 277.256,Z 268.952,A -85,B 0,C 180,E1 -17317.471,E2 -17317.471} C_VEL
LIN {X 0,Y 277.223,Z 268.952,A -85,B 0,C 180,E1 -17322.062,E2 -17322.062} C_VEL
LIN {X 0,Y 277.73,Z 271.842,A -85,B 0,C 180,E1 -17325.117,E2 -17325.117} C_VEL
LIN {X 0,Y 278.458,Z 276.073,A -85,B 0,C 180,E1 -17329.215,E2 -17329.215} C_VEL
LIN {X 0,Y 278.943,Z 280.015,A -85,B 0,C 180,E1 -17332.794,E2 -17332.794} C_VEL
LIN {X 0,Y 278.789,Z 283.138,A -85,B 0,C 180,E1 -17335.444,E2 -17335.444} C_VEL
LIN {X 0,Y 277.856,Z 288.325,A -85,B 0,C 180,E1 -17339.61,E2 -17339.61} C_VEL
LIN {X 0,Y 277.122,Z 293.132,A -85,B 0,C 180,E1 -17343.416,E2 -17343.416} C_VEL
LIN {X 0,Y 279.271,Z 301.464,A -85,B 0,C 180,E1 -17344.001,E2 -17344.001} C_VEL
LIN {X 0,Y 281.942,Z 313.448,A -85,B 0,C 180,E1 -17345.014,E2 -17345.014} C_VEL
LIN {X 0,Y 283.636,Z 324.359,A -85,B 0,C 180,E1 -17346.098,E2 -17346.098} C_VEL
LIN {X 0,Y 284.773,Z 336.587,A -85,B 0,C 180,E1 -17347.538,E2 -17347.538} C_VEL
LIN {X 0,Y 284.856,Z 342.18,A -85,B 0,C 180,E1 -17348.279,E2 -17348.279} C_VEL
LIN {X 0,Y 282.934,Z 353.06,A -85,B 0,C 180,E1 -17349.839,E2 -17349.839} C_VEL
LIN {X 0,Y 280.924,Z 363.659,A -85,B 0,C 180,E1 -17351.762,E2 -17351.762} C_VEL
LIN {X 0,Y 279.514,Z 371.599,A -85,B 0,C 180,E1 -17353.568,E2 -17353.568} C_VEL
LIN {X 0,Y 278.029,Z 379.285,A -85,B 0,C 180,E1 -17355.732,E2 -17355.732} C_VEL
LIN {X 0,Y 276.993,Z 384.554,A -85,B 0,C 180,E1 -17357.545,E2 -17357.545} C_VEL
LIN {X 0,Y 276.173,Z 389.664,A -85,B 0,C 180,E1 -17359.739,E2 -17359.739} C_VEL
LIN {X 0,Y 275.606,Z 393.634,A -85,B 0,C 180,E1 -17361.937,E2 -17361.937} C_VEL
LIN {X 0,Y 275.263,Z 397.149,A -85,B 0,C 180,E1 -17364.715,E2 -17364.715} C_VEL
LIN {X 0,Y 275.255,Z 398.966,A -85,B 0,C 180,E1 -17367.073,E2 -17367.073} C_VEL
LIN {X 0,Y 275.262,Z 399.574,A -85,B 0,C 180,E1 -17368.537,E2 -17368.537} C_VEL
LIN {X 0,Y 275.278,Z 399.788,A -85,B 0,C 180,E1 -17370,E2 -17370} C_VEL
LIN {X 0,Y 275.262,Z 399.566,A -85,B 0,C 180,E1 -17371.463,E2 -17371.463} C_VEL
LIN {X 0,Y 275.249,Z 398.953,A -85,B 0,C 180,E1 -17372.927,E2 -17372.927} C_VEL
LIN {X 0,Y 275.243,Z 397.171,A -85,B 0,C 180,E1 -17375.239,E2 -17375.239} C_VEL
LIN {X 0,Y 275.605,Z 393.595,A -85,B 0,C 180,E1 -17378.062,E2 -17378.062} C_VEL
LIN {X 0,Y 276.173,Z 389.609,A -85,B 0,C 180,E1 -17380.261,E2 -17380.261} C_VEL
LIN {X 0,Y 277.16,Z 383.482,A -85,B 0,C 180,E1 -17382.819,E2 -17382.819} C_VEL
LIN {X 0,Y 278.534,Z 376.799,A -85,B 0,C 180,E1 -17384.989,E2 -17384.989} C_VEL
LIN {X 0,Y 280.158,Z 368.507,A -85,B 0,C 180,E1 -17387.143,E2 -17387.143} C_VEL
LIN {X 0,Y 281.624,Z 360.002,A -85,B 0,C 180,E1 -17388.93,E2 -17388.93} C_VEL
LIN {X 0,Y 283.506,Z 349.499,A -85,B 0,C 180,E1 -17390.686,E2 -17390.686} C_VEL
LIN {X 0,Y 284.902,Z 340.62,A -85,B 0,C 180,E1 -17391.896,E2 -17391.896} C_VEL
LIN {X 0,Y 284.138,Z 329.407,A -85,B 0,C 180,E1 -17393.313,E2 -17393.313} C_VEL
LIN {X 0,Y 282.646,Z 317.42,A -85,B 0,C 180,E1 -17394.581,E2 -17394.581} C_VEL
LIN {X 0,Y 280.099,Z 304.904,A -85,B 0,C 180,E1 -17395.697,E2 -17395.697} C_VEL
LIN {X 0,Y 277.115,Z 293.086,A -85,B 0,C 180,E1 -17396.589,E2 -17396.589} C_VEL
LIN {X 0,Y 277.924,Z 287.883,A -85,B 0,C 180,E1 -17400.708,E2 -17400.708} C_VEL
LIN {X 0,Y 278.781,Z 283.092,A -85,B 0,C 180,E1 -17404.556,E2 -17404.556} C_VEL
LIN {X 0,Y 278.905,Z 279.959,A -85,B 0,C 180,E1 -17407.212,E2 -17407.212} C_VEL
LIN {X 0,Y 278.437,Z 276.031,A -85,B 0,C 180,E1 -17410.779,E2 -17410.779} C_VEL
LIN {X 0,Y 277.725,Z 271.787,A -85,B 0,C 180,E1 -17414.882,E2 -17414.882} C_VEL
LIN {X 0,Y 277.205,Z 268.95,A -85,B 0,C 180,E1 -17418.03,E2 -17418.03} C_VEL
LIN {X 0,Y 277.255,Z 268.949,A -85,B 0,C 180,E1 -17422.529,E2 -17422.529} C_VEL
LIN {X 0,Y 277.246,Z 268.952,A -85,B 0,C 180,E1 -17426.104,E2 -17426.104} C_VEL
LIN {X 0,Y 277.262,Z 268.949,A -85,B 0,C 180,E1 -17429.539,E2 -17429.539} C_VEL
LIN {X 0,Y 277.29,Z 268.946,A -85,B 0,C 180,E1 -17432.857,E2 -17432.857} C_VEL
LIN {X 0,Y 277.273,Z 268.95,A -85,B 0,C 180,E1 -17436.074,E2 -17436.074} C_VEL
LIN {X 0,Y 277.343,Z 268.936,A -85,B 0,C 180,E1 -17440.766,E2 -17440.766} C_VEL
LIN {X 0,Y 277.436,Z 268.926,A -85,B 0,C 180,E1 -17445.326,E2 -17445.326} C_VEL
LIN {X 0,Y 277.458,Z 268.925,A -85,B 0,C 180,E1 -17449.787,E2 -17449.787} C_VEL
LIN {X 0,Y 277.629,Z 268.9,A -85,B 0,C 180,E1 -17452.729,E2 -17452.729} C_VEL
LIN {X 0,Y 277.822,Z 268.875,A -85,B 0,C 180,E1 -17458.551,E2 -17458.551} C_VEL
LIN {X 0,Y 277.814,Z 268.879,A -85,B 0,C 180,E1 -17461.45,E2 -17461.45} C_VEL
LIN {X 0,Y 277.623,Z 268.903,A -85,B 0,C 180,E1 -17467.272,E2 -17467.272} C_VEL
LIN {X 0,Y 277.459,Z 268.922,A -85,B 0,C 180,E1 -17470.213,E2 -17470.213} C_VEL
LIN {X 0,Y 277.411,Z 268.931,A -85,B 0,C 180,E1 -17474.676,E2 -17474.676} C_VEL
LIN {X 0,Y 277.325,Z 268.939,A -85,B 0,C 180,E1 -17479.235,E2 -17479.235} C_VEL
LIN {X 0,Y 277.299,Z 268.943,A -85,B 0,C 180,E1 -17483.923,E2 -17483.923} C_VEL
LIN {X 0,Y 277.336,Z 268.937,A -85,B 0,C 180,E1 -17487.509,E2 -17487.509} C_VEL
LIN {X 0,Y 277.273,Z 268.947,A -85,B 0,C 180,E1 -17490.481,E2 -17490.481} C_VEL
LIN {X 0,Y 277.248,Z 268.951,A -85,B 0,C 180,E1 -17493.896,E2 -17493.896} C_VEL
LIN {X 0,Y 277.273,Z 268.946,A -85,B 0,C 180,E1 -17497.469,E2 -17497.469} C_VEL
LIN {X 0,Y 277.211,Z 268.954,A -85,B 0,C 180,E1 -17501.237,E2 -17501.237} C_VEL
LIN {X 0,Y 277.196,Z 268.955,A -85,B 0,C 180,E1 -17505.228,E2 -17505.228} C_VEL
LIN {X 0,Y 277.177,Z 268.96,A -85,B 0,C 180,E1 -17508.758,E2 -17508.758} C_VEL
LIN {X 0,Y 277.198,Z 268.957,A -85,B 0,C 180,E1 -17510.666,E2 -17510.666} C_VEL
LIN {X 0,Y 277.328,Z 270.186,A -85,B 0,C 180,E1 -17512.54,E2 -17512.54} C_VEL
LIN {X 0,Y 277.364,Z 271.686,A -85,B 0,C 180,E1 -17514.353,E2 -17514.353} C_VEL
LIN {X 0,Y 277.151,Z 274.722,A -85,B 0,C 180,E1 -17517.824,E2 -17517.824} C_VEL
LIN {X 0,Y 276.841,Z 277.785,A -85,B 0,C 180,E1 -17521.162,E2 -17521.162} C_VEL
LIN {X 0,Y 276.7,Z 279.967,A -85,B 0,C 180,E1 -17523.459,E2 -17523.459} C_VEL
LIN {X 0,Y 281.273,Z 294.957,A -85,B 0,C 180,E1 -17524.735,E2 -17524.735} C_VEL
LIN {X 0,Y 284.182,Z 307.093,A -85,B 0,C 180,E1 -17525.968,E2 -17525.968} C_VEL
LIN {X 0,Y 286.012,Z 317.733,A -85,B 0,C 180,E1 -17527.231,E2 -17527.231} C_VEL
LIN {X 0,Y 286.383,Z 322.429,A -85,B 0,C 180,E1 -17527.833,E2 -17527.833} C_VEL
LIN {X 0,Y 284.767,Z 333.09,A -85,B 0,C 180,E1 -17529.221,E2 -17529.221} C_VEL
LIN {X 0,Y 283.108,Z 342.784,A -85,B 0,C 180,E1 -17530.793,E2 -17530.793} C_VEL
LIN {X 0,Y 281.535,Z 351.633,A -85,B 0,C 180,E1 -17532.569,E2 -17532.569} C_VEL
LIN {X 0,Y 279.747,Z 360.251,A -85,B 0,C 180,E1 -17534.705,E2 -17534.705} C_VEL
LIN {X 0,Y 278.321,Z 367.119,A -85,B 0,C 180,E1 -17536.864,E2 -17536.864} C_VEL
LIN {X 0,Y 277.211,Z 372.616,A -85,B 0,C 180,E1 -17539.039,E2 -17539.039} C_VEL
LIN {X 0,Y 276.395,Z 376.93,A -85,B 0,C 180,E1 -17541.225,E2 -17541.225} C_VEL
LIN {X 0,Y 275.832,Z 380.359,A -85,B 0,C 180,E1 -17543.564,E2 -17543.564} C_VEL
LIN {X 0,Y 275.555,Z 382.458,A -85,B 0,C 180,E1 -17545.612,E2 -17545.612} C_VEL
LIN {X 0,Y 275.425,Z 383.45,A -85,B 0,C 180,E1 -17547.075,E2 -17547.075} C_VEL
LIN {X 0,Y 275.285,Z 384.291,A -85,B 0,C 180,E1 -17550,E2 -17550} C_VEL
LIN {X 0,Y 275.305,Z 384.099,A -85,B 0,C 180,E1 -17551.463,E2 -17551.463} C_VEL
LIN {X 0,Y 275.424,Z 383.512,A -85,B 0,C 180,E1 -17552.925,E2 -17552.925} C_VEL
LIN {X 0,Y 275.552,Z 382.545,A -85,B 0,C 180,E1 -17554.388,E2 -17554.388} C_VEL
LIN {X 0,Y 275.872,Z 380.408,A -85,B 0,C 180,E1 -17556.51,E2 -17556.51} C_VEL
LIN {X 0,Y 276.407,Z 377.127,A -85,B 0,C 180,E1 -17558.775,E2 -17558.775} C_VEL
LIN {X 0,Y 277.174,Z 372.875,A -85,B 0,C 180,E1 -17560.963,E2 -17560.963} C_VEL
LIN {X 0,Y 278.518,Z 366.433,A -85,B 0,C 180,E1 -17563.498,E2 -17563.498} C_VEL
LIN {X 0,Y 279.928,Z 359.354,A -85,B 0,C 180,E1 -17565.658,E2 -17565.658} C_VEL
LIN {X 0,Y 281.819,Z 350.527,A -85,B 0,C 180,E1 -17567.788,E2 -17567.788} C_VEL
LIN {X 0,Y 283.456,Z 341.036,A -85,B 0,C 180,E1 -17569.64,E2 -17569.64} C_VEL
LIN {X 0,Y 285.257,Z 330.155,A -85,B 0,C 180,E1 -17571.309,E2 -17571.309} C_VEL
LIN {X 0,Y 286.461,Z 321.859,A -85,B 0,C 180,E1 -17572.351,E2 -17572.351} C_VEL
LIN {X 0,Y 285.053,Z 311.693,A -85,B 0,C 180,E1 -17573.629,E2 -17573.629} C_VEL
LIN {X 0,Y 282.714,Z 300.358,A -85,B 0,C 180,E1 -17574.859,E2 -17574.859} C_VEL
LIN {X 0,Y 279.137,Z 287.755,A -85,B 0,C 180,E1 -17576.035,E2 -17576.035} C_VEL
LIN {X 0,Y 276.716,Z 279.975,A -85,B 0,C 180,E1 -17576.659,E2 -17576.659} C_VEL
LIN {X 0,Y 276.997,Z 276.361,A -85,B 0,C 180,E1 -17580.494,E2 -17580.494} C_VEL
LIN {X 0,Y 277.232,Z 273.331,A -85,B 0,C 180,E1 -17583.898,E2 -17583.898} C_VEL
LIN {X 0,Y 277.355,Z 271.675,A -85,B 0,C 180,E1 -17585.819,E2 -17585.819} C_VEL
LIN {X 0,Y 277.196,Z 268.953,A -85,B 0,C 180,E1 -17589.335,E2 -17589.335} C_VEL
LIN {X 0,Y 277.192,Z 268.952,A -85,B 0,C 180,E1 -17593.202,E2 -17593.202} C_VEL
LIN {X 0,Y 277.217,Z 268.952,A -85,B 0,C 180,E1 -17597.325,E2 -17597.325} C_VEL
LIN {X 0,Y 277.274,Z 268.946,A -85,B 0,C 180,E1 -17601.791,E2 -17601.791} C_VEL
LIN {X 0,Y 277.289,Z 268.946,A -85,B 0,C 180,E1 -17604.342,E2 -17604.342} C_VEL
LIN {X 0,Y 277.247,Z 268.952,A -85,B 0,C 180,E1 -17607.837,E2 -17607.837} C_VEL
LIN {X 0,Y 277.292,Z 268.943,A -85,B 0,C 180,E1 -17611.213,E2 -17611.213} C_VEL
LIN {X 0,Y 277.312,Z 268.94,A -85,B 0,C 180,E1 -17614.479,E2 -17614.479} C_VEL
LIN {X 0,Y 277.269,Z 268.947,A -85,B 0,C 180,E1 -17617.653,E2 -17617.653} C_VEL
LIN {X 0,Y 277.326,Z 268.938,A -85,B 0,C 180,E1 -17620.765,E2 -17620.765} C_VEL
LIN {X 0,Y 277.412,Z 268.93,A -85,B 0,C 180,E1 -17625.325,E2 -17625.325} C_VEL
LIN {X 0,Y 277.46,Z 268.922,A -85,B 0,C 180,E1 -17629.787,E2 -17629.787} C_VEL
LIN {X 0,Y 277.615,Z 268.904,A -85,B 0,C 180,E1 -17632.728,E2 -17632.728} C_VEL
LIN {X 0,Y 277.809,Z 268.88,A -85,B 0,C 180,E1 -17638.55,E2 -17638.55} C_VEL
LIN {X 0,Y 277.822,Z 268.876,A -85,B 0,C 180,E1 -17641.449,E2 -17641.449} C_VEL
LIN {X 0,Y 277.631,Z 268.9,A -85,B 0,C 180,E1 -17647.271,E2 -17647.271} C_VEL
LIN {X 0,Y 277.496,Z 268.917,A -85,B 0,C 180,E1 -17649.648,E2 -17649.648} C_VEL
LIN {X 0,Y 276.767,Z 269.011,A -85,B 0,C 180,E1 -17650.859,E2 -17650.859} C_VEL
LIN {X 0,Y 273.914,Z 269.368,A -85,B 0,C 180,E1 -17652.832,E2 -17652.832} C_VEL
LIN {X 0,Y 271.518,Z 269.666,A -85,B 0,C 180,E1 -17654.434,E2 -17654.434} C_VEL
LIN {X 0,Y 270.471,Z 269.794,A -85,B 0,C 180,E1 -17655.676,E2 -17655.676} C_VEL
LIN {X 0,Y 270.373,Z 269.805,A -85,B 0,C 180,E1 -17656.096,E2 -17656.096} C_VEL
LIN {X 0,Y 270.293,Z 269.815,A -85,B 0,C 180,E1 -17660.601,E2 -17660.601} C_VEL
LIN {X 0,Y 270.2,Z 269.826,A -85,B 0,C 180,E1 -17664.593,E2 -17664.593} C_VEL
LIN {X 0,Y 270.199,Z 269.829,A -85,B 0,C 180,E1 -17667.917,E2 -17667.917} C_VEL
LIN {X 0,Y 270.175,Z 269.832,A -85,B 0,C 180,E1 -17671.349,E2 -17671.349} C_VEL
LIN {X 0,Y 270.2,Z 269.829,A -85,B 0,C 180,E1 -17674.906,E2 -17674.906} C_VEL
LIN {X 0,Y 270.199,Z 269.829,A -85,B 0,C 180,E1 -17678.71,E2 -17678.71} C_VEL
LIN {X 0,Y 270.182,Z 269.931,A -85,B 0,C 180,E1 -17681.719,E2 -17681.719} C_VEL
LIN {X 0,Y 270.803,Z 273.505,A -85,B 0,C 180,E1 -17685.515,E2 -17685.515} C_VEL
LIN {X 0,Y 271.506,Z 277.72,A -85,B 0,C 180,E1 -17689.674,E2 -17689.674} C_VEL
LIN {X 0,Y 271.797,Z 279.815,A -85,B 0,C 180,E1 -17691.641,E2 -17691.641} C_VEL
LIN {X 0,Y 271.847,Z 282.95,A -85,B 0,C 180,E1 -17694.43,E2 -17694.43} C_VEL
LIN {X 0,Y 271.161,Z 287.093,A -85,B 0,C 180,E1 -17697.905,E2 -17697.905} C_VEL
LIN {X 0,Y 270.21,Z 292.726,A -85,B 0,C 180,E1 -17702.505,E2 -17702.505} C_VEL
LIN {X 0,Y 270.163,Z 292.934,A -85,B 0,C 180,E1 -17702.672,E2 -17702.672} C_VEL
LIN {X 0,Y 273.652,Z 306.397,A -85,B 0,C 180,E1 -17703.721,E2 -17703.721} C_VEL
LIN {X 0,Y 276.257,Z 319.742,A -85,B 0,C 180,E1 -17705,E2 -17705} C_VEL
LIN {X 0,Y 277.671,Z 332.169,A -85,B 0,C 180,E1 -17706.411,E2 -17706.411} C_VEL
LIN {X 0,Y 278.124,Z 341.98,A -85,B 0,C 180,E1 -17707.726,E2 -17707.726} C_VEL
LIN {X 0,Y 276.27,Z 352.864,A -85,B 0,C 180,E1 -17709.331,E2 -17709.331} C_VEL
LIN {X 0,Y 274.515,Z 361.745,A -85,B 0,C 180,E1 -17710.949,E2 -17710.949} C_VEL
LIN {X 0,Y 272.688,Z 371.401,A -85,B 0,C 180,E1 -17713.145,E2 -17713.145} C_VEL
LIN {X 0,Y 271.128,Z 379.086,A -85,B 0,C 180,E1 -17715.36,E2 -17715.36} C_VEL
LIN {X 0,Y 269.701,Z 386.178,A -85,B 0,C 180,E1 -17717.967,E2 -17717.967} C_VEL
LIN {X 0,Y 268.935,Z 390.899,A -85,B 0,C 180,E1 -17720.22,E2 -17720.22} C_VEL
LIN {X 0,Y 268.418,Z 394.507,A -85,B 0,C 180,E1 -17722.477,E2 -17722.477} C_VEL
LIN {X 0,Y 268.179,Z 397.144,A -85,B 0,C 180,E1 -17724.775,E2 -17724.775} C_VEL
LIN {X 0,Y 268.168,Z 398.766,A -85,B 0,C 180,E1 -17726.995,E2 -17726.995} C_VEL
LIN {X 0,Y 268.188,Z 399.375,A -85,B 0,C 180,E1 -17728.498,E2 -17728.498} C_VEL
LIN {X 0,Y 268.202,Z 399.589,A -85,B 0,C 180,E1 -17730,E2 -17730} C_VEL
LIN {X 0,Y 268.187,Z 399.367,A -85,B 0,C 180,E1 -17731.501,E2 -17731.501} C_VEL
LIN {X 0,Y 268.161,Z 398.752,A -85,B 0,C 180,E1 -17733.004,E2 -17733.004} C_VEL
LIN {X 0,Y 268.157,Z 397.169,A -85,B 0,C 180,E1 -17735.174,E2 -17735.174} C_VEL
LIN {X 0,Y 268.552,Z 393.394,A -85,B 0,C 180,E1 -17738.275,E2 -17738.275} C_VEL
LIN {X 0,Y 269.16,Z 389.408,A -85,B 0,C 180,E1 -17740.531,E2 -17740.531} C_VEL
LIN {X 0,Y 270.217,Z 383.28,A -85,B 0,C 180,E1 -17743.154,E2 -17743.154} C_VEL
LIN {X 0,Y 271.671,Z 376.597,A -85,B 0,C 180,E1 -17745.377,E2 -17745.377} C_VEL
LIN {X 0,Y 273.357,Z 368.305,A -85,B 0,C 180,E1 -17747.583,E2 -17747.583} C_VEL
LIN {X 0,Y 274.883,Z 359.798,A -85,B 0,C 180,E1 -17749.413,E2 -17749.413} C_VEL
LIN {X 0,Y 276.876,Z 349.296,A -85,B 0,C 180,E1 -17751.205,E2 -17751.205} C_VEL
LIN {X 0,Y 278.151,Z 341.759,A -85,B 0,C 180,E1 -17752.272,E2 -17752.272} C_VEL
LIN {X 0,Y 277.498,Z 331.09,A -85,B 0,C 180,E1 -17753.694,E2 -17753.694} C_VEL
LIN {X 0,Y 276.09,Z 318.847,A -85,B 0,C 180,E1 -17755.06,E2 -17755.06} C_VEL
LIN {X 0,Y 273.518,Z 305.979,A -85,B 0,C 180,E1 -17756.284,E2 -17756.284} C_VEL
LIN {X 0,Y 270.185,Z 292.888,A -85,B 0,C 180,E1 -17757.329,E2 -17757.329} C_VEL
LIN {X 0,Y 271.158,Z 287.047,A -85,B 0,C 180,E1 -17762.095,E2 -17762.095} C_VEL
LIN {X 0,Y 271.837,Z 282.887,A -85,B 0,C 180,E1 -17765.571,E2 -17765.571} C_VEL
LIN {X 0,Y 271.787,Z 279.754,A -85,B 0,C 180,E1 -17768.36,E2 -17768.36} C_VEL
LIN {X 0,Y 271.164,Z 275.566,A -85,B 0,C 180,E1 -17772.366,E2 -17772.366} C_VEL
LIN {X 0,Y 270.432,Z 271.337,A -85,B 0,C 180,E1 -17776.691,E2 -17776.691} C_VEL
LIN {X 0,Y 270.152,Z 269.829,A -85,B 0,C 180,E1 -17778.483,E2 -17778.483} C_VEL
LIN {X 0,Y 270.208,Z 269.828,A -85,B 0,C 180,E1 -17781.374,E2 -17781.374} C_VEL
LIN {X 0,Y 270.198,Z 269.828,A -85,B 0,C 180,E1 -17785.094,E2 -17785.094} C_VEL
LIN {X 0,Y 270.185,Z 269.831,A -85,B 0,C 180,E1 -17789.136,E2 -17789.136} C_VEL
LIN {X 0,Y 270.222,Z 269.83,A -85,B 0,C 180,E1 -17792.163,E2 -17792.163} C_VEL
LIN {X 0,Y 270.218,Z 269.827,A -85,B 0,C 180,E1 -17795.547,E2 -17795.547} C_VEL
LIN {X 0,Y 270.301,Z 269.816,A -85,B 0,C 180,E1 -17800.244,E2 -17800.244} C_VEL
LIN {X 0,Y 270.404,Z 269.8,A -85,B 0,C 180,E1 -17804.935,E2 -17804.935} C_VEL
LIN {X 0,Y 270.411,Z 269.802,A -85,B 0,C 180,E1 -17809.518,E2 -17809.518} C_VEL
LIN {X 0,Y 270.586,Z 269.777,A -85,B 0,C 180,E1 -17812.538,E2 -17812.538} C_VEL
LIN {X 0,Y 270.788,Z 269.751,A -85,B 0,C 180,E1 -17818.513,E2 -17818.513} C_VEL
LIN {X 0,Y 270.778,Z 269.755,A -85,B 0,C 180,E1 -17821.487,E2 -17821.487} C_VEL
LIN {X 0,Y 270.581,Z 269.779,A -85,B 0,C 180,E1 -17827.462,E2 -17827.462} C_VEL
LIN {X 0,Y 270.411,Z 269.801,A -85,B 0,C 180,E1 -17830.482,E2 -17830.482} C_VEL
LIN {X 0,Y 270.378,Z 269.805,A -85,B 0,C 180,E1 -17835.066,E2 -17835.066} C_VEL
LIN {X 0,Y 270.262,Z 269.818,A -85,B 0,C 180,E1 -17839.759,E2 -17839.759} C_VEL
LIN {X 0,Y 270.239,Z 269.824,A -85,B 0,C 180,E1 -17844.589,E2 -17844.589} C_VEL
LIN {X 0,Y 270.276,Z 269.818,A -85,B 0,C 180,E1 -17847.908,E2 -17847.908} C_VEL
LIN {X 0,Y 270.186,Z 269.828,A -85,B 0,C 180,E1 -17851.348,E2 -17851.348} C_VEL
LIN {X 0,Y 270.203,Z 269.826,A -85,B 0,C 180,E1 -17854.905,E2 -17854.905} C_VEL
LIN {X 0,Y 270.198,Z 269.826,A -85,B 0,C 180,E1 -17858.711,E2 -17858.711} C_VEL
LIN {X 0,Y 270.173,Z 269.829,A -85,B 0,C 180,E1 -17862.558,E2 -17862.558} C_VEL
LIN {X 0,Y 270.149,Z 269.833,A -85,B 0,C 180,E1 -17866.755,E2 -17866.755} C_VEL
LIN {X 0,Y 270.13,Z 269.838,A -85,B 0,C 180,E1 -17869.426,E2 -17869.426} C_VEL
LIN {X 0,Y 270.231,Z 270.381,A -85,B 0,C 180,E1 -17871.378,E2 -17871.378} C_VEL
LIN {X 0,Y 270.297,Z 273.406,A -85,B 0,C 180,E1 -17875.109,E2 -17875.109} C_VEL
LIN {X 0,Y 270.013,Z 276.95,A -85,B 0,C 180,E1 -17879.198,E2 -17879.198} C_VEL
LIN {X 0,Y 269.687,Z 280.171,A -85,B 0,C 180,E1 -17882.719,E2 -17882.719} C_VEL
LIN {X 0,Y 273.995,Z 293.822,A -85,B 0,C 180,E1 -17883.922,E2 -17883.922} C_VEL
LIN {X 0,Y 277.217,Z 306.595,A -85,B 0,C 180,E1 -17885.26,E2 -17885.26} C_VEL
LIN {X 0,Y 279.181,Z 318.115,A -85,B 0,C 180,E1 -17886.662,E2 -17886.662} C_VEL
LIN {X 0,Y 279.719,Z 322.715,A -85,B 0,C 180,E1 -17887.286,E2 -17887.286} C_VEL
LIN {X 0,Y 278.138,Z 333.294,A -85,B 0,C 180,E1 -17888.701,E2 -17888.701} C_VEL
LIN {X 0,Y 276.291,Z 343.613,A -85,B 0,C 180,E1 -17890.425,E2 -17890.425} C_VEL
LIN {X 0,Y 274.772,Z 351.835,A -85,B 0,C 180,E1 -17892.126,E2 -17892.126} C_VEL
LIN {X 0,Y 272.903,Z 360.453,A -85,B 0,C 180,E1 -17894.312,E2 -17894.312} C_VEL
LIN {X 0,Y 271.423,Z 367.321,A -85,B 0,C 180,E1 -17896.524,E2 -17896.524} C_VEL
LIN {X 0,Y 270.233,Z 372.818,A -85,B 0,C 180,E1 -17898.752,E2 -17898.752} C_VEL
LIN {X 0,Y 269.36,Z 377.131,A -85,B 0,C 180,E1 -17900.993,E2 -17900.993} C_VEL
LIN {X 0,Y 268.751,Z 380.779,A -85,B 0,C 180,E1 -17903.58,E2 -17903.58} C_VEL
LIN {X 0,Y 268.484,Z 382.658,A -85,B 0,C 180,E1 -17905.496,E2 -17905.496} C_VEL
LIN {X 0,Y 268.338,Z 383.65,A -85,B 0,C 180,E1 -17906.998,E2 -17906.998} C_VEL
LIN {X 0,Y 268.209,Z 384.49,A -85,B 0,C 180,E1 -17910,E2 -17910} C_VEL
LIN {X 0,Y 268.233,Z 384.298,A -85,B 0,C 180,E1 -17911.502,E2 -17911.502} C_VEL
LIN {X 0,Y 268.337,Z 383.711,A -85,B 0,C 180,E1 -17913.003,E2 -17913.003} C_VEL
LIN {X 0,Y 268.481,Z 382.744,A -85,B 0,C 180,E1 -17914.504,E2 -17914.504} C_VEL
LIN {X 0,Y 268.791,Z 380.826,A -85,B 0,C 180,E1 -17916.495,E2 -17916.495} C_VEL
LIN {X 0,Y 269.368,Z 377.326,A -85,B 0,C 180,E1 -17919.007,E2 -17919.007} C_VEL
LIN {X 0,Y 270.199,Z 373.073,A -85,B 0,C 180,E1 -17921.249,E2 -17921.249} C_VEL
LIN {X 0,Y 271.627,Z 366.631,A -85,B 0,C 180,E1 -17923.847,E2 -17923.847} C_VEL
LIN {X 0,Y 273.106,Z 359.551,A -85,B 0,C 180,E1 -17926.06,E2 -17926.06} C_VEL
LIN {X 0,Y 275.079,Z 350.724,A -85,B 0,C 180,E1 -17928.239,E2 -17928.239} C_VEL
LIN {X 0,Y 276.717,Z 341.545,A -85,B 0,C 180,E1 -17930.078,E2 -17930.078} C_VEL
LIN {X 0,Y 278.439,Z 331.638,A -85,B 0,C 180,E1 -17931.663,E2 -17931.663} C_VEL
LIN {X 0,Y 279.752,Z 323.536,A -85,B 0,C 180,E1 -17932.722,E2 -17932.722} C_VEL
LIN {X 0,Y 278.616,Z 314.201,A -85,B 0,C 180,E1 -17933.958,E2 -17933.958} C_VEL
LIN {X 0,Y 276.63,Z 303.876,A -85,B 0,C 180,E1 -17935.167,E2 -17935.167} C_VEL
LIN {X 0,Y 273.341,Z 291.433,A -85,B 0,C 180,E1 -17936.432,E2 -17936.432} C_VEL
LIN {X 0,Y 269.704,Z 280.17,A -85,B 0,C 180,E1 -17937.411,E2 -17937.411} C_VEL
LIN {X 0,Y 269.998,Z 276.565,A -85,B 0,C 180,E1 -17941.373,E2 -17941.373} C_VEL
LIN {X 0,Y 270.266,Z 273.53,A -85,B 0,C 180,E1 -17944.896,E2 -17944.896} C_VEL
LIN {X 0,Y 270.307,Z 272.005,A -85,B 0,C 180,E1 -17946.727,E2 -17946.727} C_VEL
LIN {X 0,Y 270.225,Z 270.416,A -85,B 0,C 180,E1 -17948.717,E2 -17948.717} C_VEL
LIN {X 0,Y 270.134,Z 269.831,A -85,B 0,C 180,E1 -17951.019,E2 -17951.019} C_VEL
LIN {X 0,Y 270.148,Z 269.833,A -85,B 0,C 180,E1 -17954.622,E2 -17954.622} C_VEL
LIN {X 0,Y 270.174,Z 269.829,A -85,B 0,C 180,E1 -17957.442,E2 -17957.442} C_VEL
LIN {X 0,Y 270.209,Z 269.825,A -85,B 0,C 180,E1 -17961.374,E2 -17961.374} C_VEL
LIN {X 0,Y 270.205,Z 269.826,A -85,B 0,C 180,E1 -17965.095,E2 -17965.095} C_VEL
LIN {X 0,Y 270.203,Z 269.824,A -85,B 0,C 180,E1 -17969.131,E2 -17969.131} C_VEL
LIN {X 0,Y 270.267,Z 269.817,A -85,B 0,C 180,E1 -17972.146,E2 -17972.146} C_VEL
LIN {X 0,Y 270.241,Z 269.823,A -85,B 0,C 180,E1 -17975.537,E2 -17975.537} C_VEL
LIN {X 0,Y 270.263,Z 269.818,A -85,B 0,C 180,E1 -17980.241,E2 -17980.241} C_VEL
LIN {X 0,Y 270.38,Z 269.805,A -85,B 0,C 180,E1 -17984.934,E2 -17984.934} C_VEL
LIN {X 0,Y 270.413,Z 269.801,A -85,B 0,C 180,E1 -17989.518,E2 -17989.518} C_VEL
LIN {X 0,Y 270.574,Z 269.78,A -85,B 0,C 180,E1 -17992.538,E2 -17992.538} C_VEL
LIN {X 0,Y 270.774,Z 269.757,A -85,B 0,C 180,E1 -17998.513,E2 -17998.513} C_VEL
LIN {X 0,Y 270.788,Z 269.752,A -85,B 0,C 180,E1 -18001.487,E2 -18001.487} C_VEL
LIN {X 0,Y 270.587,Z 269.777,A -85,B 0,C 180,E1 -18007.462,E2 -18007.462} C_VEL
LIN {X 0,Y 270.412,Z 269.803,A -85,B 0,C 180,E1 -18010.482,E2 -18010.482} C_VEL
LIN {X 0,Y 270.405,Z 269.8,A -85,B 0,C 180,E1 -18015.064,E2 -18015.064} C_VEL
LIN {X 0,Y 270.373,Z 269.805,A -85,B 0,C 180,E1 -18016.096,E2 -18016.096} C_VEL
LIN {X 0,Y 269.652,Z 269.895,A -85,B 0,C 180,E1 -18017.34,E2 -18017.34} C_VEL
LIN {X 0,Y 266.718,Z 270.26,A -85,B 0,C 180,E1 -18019.365,E2 -18019.365} C_VEL
LIN {X 0,Y 264.252,Z 270.567,A -85,B 0,C 180,E1 -18021.011,E2 -18021.011} C_VEL
LIN {X 0,Y 263.198,Z 270.701,A -85,B 0,C 180,E1 -18022.289,E2 -18022.289} C_VEL
LIN {X 0,Y 263.114,Z 270.708,A -85,B 0,C 180,E1 -18022.722,E2 -18022.722} C_VEL
LIN {X 0,Y 263.138,Z 270.706,A -85,B 0,C 180,E1 -18025.299,E2 -18025.299} C_VEL
LIN {X 0,Y 263.135,Z 270.707,A -85,B 0,C 180,E1 -18028.735,E2 -18028.735} C_VEL
LIN {X 0,Y 263.13,Z 270.709,A -85,B 0,C 180,E1 -18032.289,E2 -18032.289} C_VEL
LIN {X 0,Y 263.177,Z 270.704,A -85,B 0,C 180,E1 -18036.761,E2 -18036.761} C_VEL
LIN {X 0,Y 263.149,Z 270.816,A -85,B 0,C 180,E1 -18041.173,E2 -18041.173} C_VEL
LIN {X 0,Y 263.557,Z 273.312,A -85,B 0,C 180,E1 -18043.947,E2 -18043.947} C_VEL
LIN {X 0,Y 264.279,Z 277.307,A -85,B 0,C 180,E1 -18048.126,E2 -18048.126} C_VEL
LIN {X 0,Y 264.757,Z 280.668,A -85,B 0,C 180,E1 -18051.405,E2 -18051.405} C_VEL
LIN {X 0,Y 264.818,Z 283.787,A -85,B 0,C 180,E1 -18054.277,E2 -18054.277} C_VEL
LIN {X 0,Y 264.311,Z 286.894,A -85,B 0,C 180,E1 -18056.969,E2 -18056.969} C_VEL
LIN {X 0,Y 263.26,Z 292.72,A -85,B 0,C 180,E1 -18061.885,E2 -18061.885} C_VEL
LIN {X 0,Y 266.835,Z 306.458,A -85,B 0,C 180,E1 -18063.014,E2 -18063.014} C_VEL
LIN {X 0,Y 269.206,Z 318.323,A -85,B 0,C 180,E1 -18064.188,E2 -18064.188} C_VEL
LIN {X 0,Y 270.626,Z 329.284,A -85,B 0,C 180,E1 -18065.448,E2 -18065.448} C_VEL
LIN {X 0,Y 271.365,Z 340.624,A -85,B 0,C 180,E1 -18066.976,E2 -18066.976} C_VEL
LIN {X 0,Y 270.982,Z 345.684,A -85,B 0,C 180,E1 -18067.709,E2 -18067.709} C_VEL
LIN {X 0,Y 268.93,Z 355.847,A -85,B 0,C 180,E1 -18069.341,E2 -18069.341} C_VEL
LIN {X 0,Y 267.043,Z 365.171,A -85,B 0,C 180,E1 -18071.232,E2 -18071.232} C_VEL
LIN {X 0,Y 265.289,Z 373.938,A -85,B 0,C 180,E1 -18073.454,E2 -18073.454} C_VEL
LIN {X 0,Y 263.76,Z 381.125,A -85,B 0,C 180,E1 -18075.731,E2 -18075.731} C_VEL
LIN {X 0,Y 262.712,Z 385.978,A -85,B 0,C 180,E1 -18077.642,E2 -18077.642} C_VEL
LIN {X 0,Y 261.897,Z 390.699,A -85,B 0,C 180,E1 -18079.954,E2 -18079.954} C_VEL
LIN {X 0,Y 261.353,Z 394.308,A -85,B 0,C 180,E1 -18082.273,E2 -18082.273} C_VEL
LIN {X 0,Y 261.085,Z 397.162,A -85,B 0,C 180,E1 -18084.863,E2 -18084.863} C_VEL
LIN {X 0,Y 261.063,Z 398.566,A -85,B 0,C 180,E1 -18086.913,E2 -18086.913} C_VEL
LIN {X 0,Y 261.115,Z 399.176,A -85,B 0,C 180,E1 -18088.458,E2 -18088.458} C_VEL
LIN {X 0,Y 261.128,Z 399.39,A -85,B 0,C 180,E1 -18090,E2 -18090} C_VEL
LIN {X 0,Y 261.114,Z 399.167,A -85,B 0,C 180,E1 -18091.542,E2 -18091.542} C_VEL
LIN {X 0,Y 261.056,Z 398.552,A -85,B 0,C 180,E1 -18093.086,E2 -18093.086} C_VEL
LIN {X 0,Y 261.054,Z 397.21,A -85,B 0,C 180,E1 -18095.059,E2 -18095.059} C_VEL
LIN {X 0,Y 261.339,Z 394.267,A -85,B 0,C 180,E1 -18097.727,E2 -18097.727} C_VEL
LIN {X 0,Y 261.897,Z 390.641,A -85,B 0,C 180,E1 -18100.045,E2 -18100.045} C_VEL
LIN {X 0,Y 262.711,Z 385.903,A -85,B 0,C 180,E1 -18102.358,E2 -18102.358} C_VEL
LIN {X 0,Y 264.236,Z 378.797,A -85,B 0,C 180,E1 -18105.03,E2 -18105.03} C_VEL
LIN {X 0,Y 265.917,Z 371.083,A -85,B 0,C 180,E1 -18107.297,E2 -18107.297} C_VEL
LIN {X 0,Y 267.436,Z 363.189,A -85,B 0,C 180,E1 -18109.176,E2 -18109.176} C_VEL
LIN {X 0,Y 269.381,Z 353.558,A -85,B 0,C 180,E1 -18111.022,E2 -18111.022} C_VEL
LIN {X 0,Y 271.356,Z 342.877,A -85,B 0,C 180,E1 -18112.66,E2 -18112.66} C_VEL
LIN {X 0,Y 270.792,Z 331.948,A -85,B 0,C 180,E1 -18114.194,E2 -18114.194} C_VEL
LIN {X 0,Y 269.546,Z 320.334,A -85,B 0,C 180,E1 -18115.557,E2 -18115.557} C_VEL
LIN {X 0,Y 267.034,Z 307.36,A -85,B 0,C 180,E1 -18116.863,E2 -18116.863} C_VEL
LIN {X 0,Y 263.561,Z 294.493,A -85,B 0,C 180,E1 -18117.961,E2 -18117.961} C_VEL
LIN {X 0,Y 263.26,Z 292.711,A -85,B 0,C 180,E1 -18118.086,E2 -18118.086} C_VEL
LIN {X 0,Y 264.308,Z 286.845,A -85,B 0,C 180,E1 -18123.031,E2 -18123.031} C_VEL
LIN {X 0,Y 264.809,Z 283.734,A -85,B 0,C 180,E1 -18125.724,E2 -18125.724} C_VEL
LIN {X 0,Y 264.741,Z 280.589,A -85,B 0,C 180,E1 -18128.598,E2 -18128.598} C_VEL
LIN {X 0,Y 264.263,Z 277.263,A -85,B 0,C 180,E1 -18131.871,E2 -18131.871} C_VEL
LIN {X 0,Y 263.532,Z 273.209,A -85,B 0,C 180,E1 -18136.102,E2 -18136.102} C_VEL
LIN {X 0,Y 263.106,Z 270.711,A -85,B 0,C 180,E1 -18139.039,E2 -18139.039} C_VEL
LIN {X 0,Y 263.176,Z 270.703,A -85,B 0,C 180,E1 -18143.239,E2 -18143.239} C_VEL
LIN {X 0,Y 263.129,Z 270.711,A -85,B 0,C 180,E1 -18147.711,E2 -18147.711} C_VEL
LIN {X 0,Y 263.148,Z 270.709,A -85,B 0,C 180,E1 -18151.805,E2 -18151.805} C_VEL
LIN {X 0,Y 263.138,Z 270.709,A -85,B 0,C 180,E1 -18156.383,E2 -18156.383} C_VEL
LIN {X 0,Y 263.25,Z 270.695,A -85,B 0,C 180,E1 -18159.692,E2 -18159.692} C_VEL
LIN {X 0,Y 263.352,Z 270.679,A -85,B 0,C 180,E1 -18164.522,E2 -18164.522} C_VEL
LIN {X 0,Y 263.354,Z 270.68,A -85,B 0,C 180,E1 -18169.234,E2 -18169.234} C_VEL
LIN {X 0,Y 263.545,Z 270.654,A -85,B 0,C 180,E1 -18172.338,E2 -18172.338} C_VEL
LIN {X 0,Y 263.752,Z 270.627,A -85,B 0,C 180,E1 -18178.473,E2 -18178.473} C_VEL
LIN {X 0,Y 263.741,Z 270.631,A -85,B 0,C 180,E1 -18181.527,E2 -18181.527} C_VEL
LIN {X 0,Y 263.541,Z 270.655,A -85,B 0,C 180,E1 -18187.663,E2 -18187.663} C_VEL
LIN {X 0,Y 263.351,Z 270.683,A -85,B 0,C 180,E1 -18190.767,E2 -18190.767} C_VEL
LIN {X 0,Y 263.325,Z 270.682,A -85,B 0,C 180,E1 -18195.48,E2 -18195.48} C_VEL
LIN {X 0,Y 263.239,Z 270.696,A -85,B 0,C 180,E1 -18200.309,E2 -18200.309} C_VEL
LIN {X 0,Y 263.195,Z 270.699,A -85,B 0,C 180,E1 -18205.293,E2 -18205.293} C_VEL
LIN {X 0,Y 263.185,Z 270.7,A -85,B 0,C 180,E1 -18208.729,E2 -18208.729} C_VEL
LIN {X 0,Y 263.134,Z 270.71,A -85,B 0,C 180,E1 -18212.288,E2 -18212.288} C_VEL
LIN {X 0,Y 263.177,Z 270.704,A -85,B 0,C 180,E1 -18215.98,E2 -18215.98} C_VEL
LIN {X 0,Y 263.107,Z 270.71,A -85,B 0,C 180,E1 -18219.873,E2 -18219.873} C_VEL
LIN {X 0,Y 263.104,Z 270.712,A -85,B 0,C 180,E1 -18223.988,E2 -18223.988} C_VEL
LIN {X 0,Y 263.076,Z 270.716,A -85,B 0,C 180,E1 -18228.097,E2 -18228.097} C_VEL
LIN {X 0,Y 263.089,Z 270.715,A -85,B 0,C 180,E1 -18230.125,E2 -18230.125} C_VEL
LIN {X 0,Y 263.294,Z 272.931,A -85,B 0,C 180,E1 -18233.205,E2 -18233.205} C_VEL
LIN {X 0,Y 263.259,Z 275.122,A -85,B 0,C 180,E1 -18235.901,E2 -18235.901} C_VEL
LIN {X 0,Y 262.928,Z 278.199,A -85,B 0,C 180,E1 -18239.478,E2 -18239.478} C_VEL
LIN {X 0,Y 262.695,Z 280.381,A -85,B 0,C 180,E1 -18241.919,E2 -18241.919} C_VEL
LIN {X 0,Y 263.655,Z 283.484,A -85,B 0,C 180,E1 -18242.195,E2 -18242.195} C_VEL
LIN {X 0,Y 267.665,Z 295.928,A -85,B 0,C 180,E1 -18243.389,E2 -18243.389} C_VEL
LIN {X 0,Y 270.644,Z 307.99,A -85,B 0,C 180,E1 -18244.728,E2 -18244.728} C_VEL
LIN {X 0,Y 272.454,Z 318.929,A -85,B 0,C 180,E1 -18246.127,E2 -18246.127} C_VEL
LIN {X 0,Y 273.004,Z 324.506,A -85,B 0,C 180,E1 -18246.917,E2 -18246.917} C_VEL
LIN {X 0,Y 271.136,Z 335.836,A -85,B 0,C 180,E1 -18248.523,E2 -18248.523} C_VEL
LIN {X 0,Y 269.385,Z 345.15,A -85,B 0,C 180,E1 -18250.175,E2 -18250.175} C_VEL
LIN {X 0,Y 267.666,Z 353.634,A -85,B 0,C 180,E1 -18252.03,E2 -18252.03} C_VEL
LIN {X 0,Y 265.792,Z 361.882,A -85,B 0,C 180,E1 -18254.275,E2 -18254.275} C_VEL
LIN {X 0,Y 264.265,Z 368.524,A -85,B 0,C 180,E1 -18256.544,E2 -18256.544} C_VEL
LIN {X 0,Y 262.91,Z 374.606,A -85,B 0,C 180,E1 -18259.215,E2 -18259.215} C_VEL
LIN {X 0,Y 262.118,Z 378.553,A -85,B 0,C 180,E1 -18261.52,E2 -18261.52} C_VEL
LIN {X 0,Y 261.601,Z 381.466,A -85,B 0,C 180,E1 -18263.831,E2 -18263.831} C_VEL
LIN {X 0,Y 261.398,Z 382.859,A -85,B 0,C 180,E1 -18265.374,E2 -18265.374} C_VEL
LIN {X 0,Y 261.255,Z 383.85,A -85,B 0,C 180,E1 -18266.916,E2 -18266.916} C_VEL
LIN {X 0,Y 261.135,Z 384.689,A -85,B 0,C 180,E1 -18270,E2 -18270} C_VEL
LIN {X 0,Y 261.163,Z 384.496,A -85,B 0,C 180,E1 -18271.542,E2 -18271.542} C_VEL
LIN {X 0,Y 261.254,Z 383.91,A -85,B 0,C 180,E1 -18273.084,E2 -18273.084} C_VEL
LIN {X 0,Y 261.621,Z 381.587,A -85,B 0,C 180,E1 -18276.169,E2 -18276.169} C_VEL
LIN {X 0,Y 262.16,Z 378.719,A -85,B 0,C 180,E1 -18278.479,E2 -18278.479} C_VEL
LIN {X 0,Y 262.893,Z 374.831,A -85,B 0,C 180,E1 -18280.786,E2 -18280.786} C_VEL
LIN {X 0,Y 264.022,Z 369.812,A -85,B 0,C 180,E1 -18283.077,E2 -18283.077} C_VEL
LIN {X 0,Y 265.399,Z 363.491,A -85,B 0,C 180,E1 -18285.356,E2 -18285.356} C_VEL
LIN {X 0,Y 267.256,Z 355.575,A -85,B 0,C 180,E1 -18287.603,E2 -18287.603} C_VEL
LIN {X 0,Y 269.022,Z 347.505,A -85,B 0,C 180,E1 -18289.456,E2 -18289.456} C_VEL
LIN {X 0,Y 270.829,Z 337.662,A -85,B 0,C 180,E1 -18291.303,E2 -18291.303} C_VEL
LIN {X 0,Y 272.576,Z 327.966,A -85,B 0,C 180,E1 -18292.753,E2 -18292.753} C_VEL
LIN {X 0,Y 273.073,Z 323.879,A -85,B 0,C 180,E1 -18293.29,E2 -18293.29} C_VEL
LIN {X 0,Y 271.497,Z 312.473,A -85,B 0,C 180,E1 -18294.847,E2 -18294.847} C_VEL
LIN {X 0,Y 269.06,Z 301.147,A -85,B 0,C 180,E1 -18296.183,E2 -18296.183} C_VEL
LIN {X 0,Y 265.468,Z 288.592,A -85,B 0,C 180,E1 -18297.46,E2 -18297.46} C_VEL
LIN {X 0,Y 262.769,Z 280.941,A -85,B 0,C 180,E1 -18298.159,E2 -18298.159} C_VEL
LIN {X 0,Y 262.701,Z 280.351,A -85,B 0,C 180,E1 -18298.25,E2 -18298.25} C_VEL
LIN {X 0,Y 263.038,Z 276.769,A -85,B 0,C 180,E1 -18302.302,E2 -18302.302} C_VEL
LIN {X 0,Y 263.282,Z 273.71,A -85,B 0,C 180,E1 -18305.963,E2 -18305.963} C_VEL
LIN {X 0,Y 263.089,Z 270.709,A -85,B 0,C 180,E1 -18309.876,E2 -18309.876} C_VEL
LIN {X 0,Y 263.1,Z 270.709,A -85,B 0,C 180,E1 -18313.989,E2 -18313.989} C_VEL
LIN {X 0,Y 263.126,Z 270.71,A -85,B 0,C 180,E1 -18318.407,E2 -18318.407} C_VEL
LIN {X 0,Y 263.196,Z 270.698,A -85,B 0,C 180,E1 -18323.233,E2 -18323.233} C_VEL
LIN {X 0,Y 263.17,Z 270.703,A -85,B 0,C 180,E1 -18325.888,E2 -18325.888} C_VEL
LIN {X 0,Y 263.153,Z 270.703,A -85,B 0,C 180,E1 -18329.507,E2 -18329.507} C_VEL
LIN {X 0,Y 263.194,Z 270.696,A -85,B 0,C 180,E1 -18333.003,E2 -18333.003} C_VEL
LIN {X 0,Y 263.157,Z 270.7,A -85,B 0,C 180,E1 -18336.384,E2 -18336.384} C_VEL
LIN {X 0,Y 263.241,Z 270.695,A -85,B 0,C 180,E1 -18339.691,E2 -18339.691} C_VEL
LIN {X 0,Y 263.326,Z 270.682,A -85,B 0,C 180,E1 -18344.52,E2 -18344.52} C_VEL
LIN {X 0,Y 263.355,Z 270.682,A -85,B 0,C 180,E1 -18349.234,E2 -18349.234} C_VEL
LIN {X 0,Y 263.536,Z 270.656,A -85,B 0,C 180,E1 -18352.337,E2 -18352.337} C_VEL
LIN {X 0,Y 263.738,Z 270.633,A -85,B 0,C 180,E1 -18358.473,E2 -18358.473} C_VEL
LIN {X 0,Y 263.753,Z 270.629,A -85,B 0,C 180,E1 -18361.527,E2 -18361.527} C_VEL
LIN {X 0,Y 263.547,Z 270.654,A -85,B 0,C 180,E1 -18367.662,E2 -18367.662} C_VEL
LIN {X 0,Y 263.355,Z 270.681,A -85,B 0,C 180,E1 -18370.766,E2 -18370.766} C_VEL
LIN {X 0,Y 263.354,Z 270.678,A -85,B 0,C 180,E1 -18375.478,E2 -18375.478} C_VEL
LIN {X 0,Y 263.265,Z 270.693,A -85,B 0,C 180,E1 -18380.307,E2 -18380.307} C_VEL
LIN {X 0,Y 263.114,Z 270.708,A -85,B 0,C 180,E1 -18382.722,E2 -18382.722} C_VEL
LIN {X 0,Y 262.446,Z 270.795,A -85,B 0,C 180,E1 -18383.999,E2 -18383.999} C_VEL
LIN {X 0,Y 259.592,Z 271.148,A -85,B 0,C 180,E1 -18386.08,E2 -18386.08} C_VEL
LIN {X 0,Y 257.171,Z 271.453,A -85,B 0,C 180,E1 -18387.773,E2 -18387.773} C_VEL
LIN {X 0,Y 256.137,Z 271.579,A -85,B 0,C 180,E1 -18389.086,E2 -18389.086} C_VEL
LIN {X 0,Y 256.056,Z 271.591,A -85,B 0,C 180,E1 -18389.53,E2 -18389.53} C_VEL
LIN {X 0,Y 256.068,Z 271.59,A -85,B 0,C 180,E1 -18393.293,E2 -18393.293} C_VEL
LIN {X 0,Y 256.112,Z 271.585,A -85,B 0,C 180,E1 -18397.269,E2 -18397.269} C_VEL
LIN {X 0,Y 256.067,Z 271.71,A -85,B 0,C 180,E1 -18400.613,E2 -18400.613} C_VEL
LIN {X 0,Y 256.807,Z 275.897,A -85,B 0,C 180,E1 -18405.36,E2 -18405.36} C_VEL
LIN {X 0,Y 257.398,Z 279.415,A -85,B 0,C 180,E1 -18409.057,E2 -18409.057} C_VEL
LIN {X 0,Y 257.789,Z 282.646,A -85,B 0,C 180,E1 -18412.243,E2 -18412.243} C_VEL
LIN {X 0,Y 257.682,Z 285.671,A -85,B 0,C 180,E1 -18415.057,E2 -18415.057} C_VEL
LIN {X 0,Y 256.859,Z 289.763,A -85,B 0,C 180,E1 -18418.677,E2 -18418.677} C_VEL
LIN {X 0,Y 256.354,Z 292.658,A -85,B 0,C 180,E1 -18421.073,E2 -18421.073} C_VEL
LIN {X 0,Y 259.968,Z 306.069,A -85,B 0,C 180,E1 -18422.228,E2 -18422.228} C_VEL
LIN {X 0,Y 262.549,Z 318.933,A -85,B 0,C 180,E1 -18423.56,E2 -18423.56} C_VEL
LIN {X 0,Y 263.942,Z 329.784,A -85,B 0,C 180,E1 -18424.867,E2 -18424.867} C_VEL
LIN {X 0,Y 264.61,Z 340.544,A -85,B 0,C 180,E1 -18426.371,E2 -18426.371} C_VEL
LIN {X 0,Y 264.408,Z 345.487,A -85,B 0,C 180,E1 -18427.124,E2 -18427.124} C_VEL
LIN {X 0,Y 262.307,Z 355.65,A -85,B 0,C 180,E1 -18428.795,E2 -18428.795} C_VEL
LIN {X 0,Y 260.332,Z 364.807,A -85,B 0,C 180,E1 -18430.688,E2 -18430.688} C_VEL
LIN {X 0,Y 258.448,Z 373.739,A -85,B 0,C 180,E1 -18433.003,E2 -18433.003} C_VEL
LIN {X 0,Y 256.862,Z 380.926,A -85,B 0,C 180,E1 -18435.339,E2 -18435.339} C_VEL
LIN {X 0,Y 255.738,Z 385.778,A -85,B 0,C 180,E1 -18437.3,E2 -18437.3} C_VEL
LIN {X 0,Y 254.865,Z 390.499,A -85,B 0,C 180,E1 -18439.674,E2 -18439.674} C_VEL
LIN {X 0,Y 254.312,Z 394.108,A -85,B 0,C 180,E1 -18442.057,E2 -18442.057} C_VEL
LIN {X 0,Y 253.99,Z 397.168,A -85,B 0,C 180,E1 -18444.961,E2 -18444.961} C_VEL
LIN {X 0,Y 253.963,Z 398.366,A -85,B 0,C 180,E1 -18446.827,E2 -18446.827} C_VEL
LIN {X 0,Y 254.021,Z 398.977,A -85,B 0,C 180,E1 -18448.414,E2 -18448.414} C_VEL
LIN {X 0,Y 254.055,Z 399.191,A -85,B 0,C 180,E1 -18450,E2 -18450} C_VEL
LIN {X 0,Y 254.019,Z 398.967,A -85,B 0,C 180,E1 -18451.585,E2 -18451.585} C_VEL
LIN {X 0,Y 253.956,Z 398.352,A -85,B 0,C 180,E1 -18453.173,E2 -18453.173} C_VEL
LIN {X 0,Y 253.957,Z 397.21,A -85,B 0,C 180,E1 -18454.953,E2 -18454.953} C_VEL
LIN {X 0,Y 254.303,Z 394.067,A -85,B 0,C 180,E1 -18457.943,E2 -18457.943} C_VEL
LIN {X 0,Y 254.865,Z 390.438,A -85,B 0,C 180,E1 -18460.325,E2 -18460.325} C_VEL
LIN {X 0,Y 255.737,Z 385.701,A -85,B 0,C 180,E1 -18462.7,E2 -18462.7} C_VEL
LIN {X 0,Y 257.371,Z 378.595,A -85,B 0,C 180,E1 -18465.441,E2 -18465.441} C_VEL
LIN {X 0,Y 259.106,Z 371.013,A -85,B 0,C 180,E1 -18467.73,E2 -18467.73} C_VEL
LIN {X 0,Y 260.714,Z 362.986,A -85,B 0,C 180,E1 -18469.691,E2 -18469.691} C_VEL
LIN {X 0,Y 262.751,Z 353.355,A -85,B 0,C 180,E1 -18471.579,E2 -18471.579} C_VEL
LIN {X 0,Y 264.573,Z 343.967,A -85,B 0,C 180,E1 -18473.067,E2 -18473.067} C_VEL
LIN {X 0,Y 264.186,Z 333.805,A -85,B 0,C 180,E1 -18474.569,E2 -18474.569} C_VEL
LIN {X 0,Y 263.088,Z 322.455,A -85,B 0,C 180,E1 -18475.999,E2 -18475.999} C_VEL
LIN {X 0,Y 260.965,Z 310.684,A -85,B 0,C 180,E1 -18477.287,E2 -18477.287} C_VEL
LIN {X 0,Y 257.753,Z 297.893,A -85,B 0,C 180,E1 -18478.473,E2 -18478.473} C_VEL
LIN {X 0,Y 256.325,Z 292.512,A -85,B 0,C 180,E1 -18478.9,E2 -18478.9} C_VEL
LIN {X 0,Y 257.283,Z 287.674,A -85,B 0,C 180,E1 -18483.115,E2 -18483.115} C_VEL
LIN {X 0,Y 257.691,Z 285.437,A -85,B 0,C 180,E1 -18485.096,E2 -18485.096} C_VEL
LIN {X 0,Y 257.774,Z 282.557,A -85,B 0,C 180,E1 -18487.753,E2 -18487.753} C_VEL
LIN {X 0,Y 257.382,Z 279.35,A -85,B 0,C 180,E1 -18490.945,E2 -18490.945} C_VEL
LIN {X 0,Y 256.794,Z 275.854,A -85,B 0,C 180,E1 -18494.637,E2 -18494.637} C_VEL
LIN {X 0,Y 256.06,Z 271.593,A -85,B 0,C 180,E1 -18499.483,E2 -18499.483} C_VEL
LIN {X 0,Y 256.126,Z 271.581,A -85,B 0,C 180,E1 -18502.867,E2 -18502.867} C_VEL
LIN {X 0,Y 256.066,Z 271.592,A -85,B 0,C 180,E1 -18506.707,E2 -18506.707} C_VEL
LIN {X 0,Y 256.055,Z 271.594,A -85,B 0,C 180,E1 -18510.393,E2 -18510.393} C_VEL
LIN {X 0,Y 256.083,Z 271.591,A -85,B 0,C 180,E1 -18513.953,E2 -18513.953} C_VEL
LIN {X 0,Y 256.074,Z 271.588,A -85,B 0,C 180,E1 -18517.404,E2 -18517.404} C_VEL
LIN {X 0,Y 256.181,Z 271.573,A -85,B 0,C 180,E1 -18520.78,E2 -18520.78} C_VEL
LIN {X 0,Y 256.301,Z 271.559,A -85,B 0,C 180,E1 -18524.085,E2 -18524.085} C_VEL
LIN {X 0,Y 256.297,Z 271.558,A -85,B 0,C 180,E1 -18528.933,E2 -18528.933} C_VEL
LIN {X 0,Y 256.505,Z 271.532,A -85,B 0,C 180,E1 -18532.126,E2 -18532.126} C_VEL
LIN {X 0,Y 256.499,Z 271.534,A -85,B 0,C 180,E1 -18536.859,E2 -18536.859} C_VEL
LIN {X 0,Y 256.75,Z 271.502,A -85,B 0,C 180,E1 -18540,E2 -18540} C_VEL
LIN {X 0,Y 256.46,Z 271.541,A -85,B 0,C 180,E1 -18543.142,E2 -18543.142} C_VEL
LIN {X 0,Y 256.502,Z 271.531,A -85,B 0,C 180,E1 -18547.874,E2 -18547.874} C_VEL
LIN {X 0,Y 256.292,Z 271.56,A -85,B 0,C 180,E1 -18551.067,E2 -18551.067} C_VEL
LIN {X 0,Y 256.26,Z 271.562,A -85,B 0,C 180,E1 -18555.918,E2 -18555.918} C_VEL
LIN {X 0,Y 256.15,Z 271.577,A -85,B 0,C 180,E1 -18560.897,E2 -18560.897} C_VEL
LIN {X 0,Y 256.172,Z 271.574,A -85,B 0,C 180,E1 -18565.13,E2 -18565.13} C_VEL
LIN {X 0,Y 256.118,Z 271.58,A -85,B 0,C 180,E1 -18569.599,E2 -18569.599} C_VEL
LIN {X 0,Y 256.078,Z 271.586,A -85,B 0,C 180,E1 -18573.292,E2 -18573.292} C_VEL
LIN {X 0,Y 256.123,Z 271.58,A -85,B 0,C 180,E1 -18577.273,E2 -18577.273} C_VEL
LIN {X 0,Y 256.055,Z 271.589,A -85,B 0,C 180,E1 -18581.204,E2 -18581.204} C_VEL
LIN {X 0,Y 256.038,Z 271.593,A -85,B 0,C 180,E1 -18585.535,E2 -18585.535} C_VEL
LIN {X 0,Y 256.013,Z 271.597,A -85,B 0,C 180,E1 -18588.788,E2 -18588.788} C_VEL
LIN {X 0,Y 256.097,Z 271.818,A -85,B 0,C 180,E1 -18590.211,E2 -18590.211} C_VEL
LIN {X 0,Y 256.255,Z 273.809,A -85,B 0,C 180,E1 -18592.889,E2 -18592.889} C_VEL
LIN {X 0,Y 256.131,Z 276.857,A -85,B 0,C 180,E1 -18596.717,E2 -18596.717} C_VEL
LIN {X 0,Y 255.755,Z 279.958,A -85,B 0,C 180,E1 -18600.355,E2 -18600.355} C_VEL
LIN {X 0,Y 255.71,Z 280.701,A -85,B 0,C 180,E1 -18601.107,E2 -18601.107} C_VEL
LIN {X 0,Y 256.702,Z 283.754,A -85,B 0,C 180,E1 -18601.375,E2 -18601.375} C_VEL
LIN {X 0,Y 260.758,Z 295.834,A -85,B 0,C 180,E1 -18602.603,E2 -18602.603} C_VEL
LIN {X 0,Y 263.792,Z 308.158,A -85,B 0,C 180,E1 -18604.018,E2 -18604.018} C_VEL
LIN {X 0,Y 265.788,Z 319.781,A -85,B 0,C 180,E1 -18605.575,E2 -18605.575} C_VEL
LIN {X 0,Y 266.283,Z 326.113,A -85,B 0,C 180,E1 -18606.503,E2 -18606.503} C_VEL
LIN {X 0,Y 264.356,Z 337.194,A -85,B 0,C 180,E1 -18608.149,E2 -18608.149} C_VEL
LIN {X 0,Y 262.357,Z 347.157,A -85,B 0,C 180,E1 -18610.029,E2 -18610.029} C_VEL
LIN {X 0,Y 260.266,Z 356.793,A -85,B 0,C 180,E1 -18612.315,E2 -18612.315} C_VEL
LIN {X 0,Y 258.349,Z 364.479,A -85,B 0,C 180,E1 -18614.619,E2 -18614.619} C_VEL
LIN {X 0,Y 256.716,Z 371.529,A -85,B 0,C 180,E1 -18617.349,E2 -18617.349} C_VEL
LIN {X 0,Y 255.604,Z 376.224,A -85,B 0,C 180,E1 -18619.705,E2 -18619.705} C_VEL
LIN {X 0,Y 254.885,Z 379.813,A -85,B 0,C 180,E1 -18622.076,E2 -18622.076} C_VEL
LIN {X 0,Y 254.514,Z 381.776,A -85,B 0,C 180,E1 -18623.767,E2 -18623.767} C_VEL
LIN {X 0,Y 254.174,Z 384.05,A -85,B 0,C 180,E1 -18626.83,E2 -18626.83} C_VEL
LIN {X 0,Y 254.094,Z 384.659,A -85,B 0,C 180,E1 -18628.415,E2 -18628.415} C_VEL
LIN {X 0,Y 254.063,Z 384.888,A -85,B 0,C 180,E1 -18630,E2 -18630} C_VEL
LIN {X 0,Y 254.094,Z 384.695,A -85,B 0,C 180,E1 -18631.585,E2 -18631.585} C_VEL
LIN {X 0,Y 254.173,Z 384.11,A -85,B 0,C 180,E1 -18633.17,E2 -18633.17} C_VEL
LIN {X 0,Y 254.566,Z 381.786,A -85,B 0,C 180,E1 -18636.34,E2 -18636.34} C_VEL
LIN {X 0,Y 255.13,Z 378.918,A -85,B 0,C 180,E1 -18638.714,E2 -18638.714} C_VEL
LIN {X 0,Y 255.926,Z 375.03,A -85,B 0,C 180,E1 -18641.083,E2 -18641.083} C_VEL
LIN {X 0,Y 257.11,Z 370.01,A -85,B 0,C 180,E1 -18643.435,E2 -18643.435} C_VEL
LIN {X 0,Y 258.56,Z 363.689,A -85,B 0,C 180,E1 -18645.772,E2 -18645.772} C_VEL
LIN {X 0,Y 260.493,Z 355.772,A -85,B 0,C 180,E1 -18648.075,E2 -18648.075} C_VEL
LIN {X 0,Y 262.33,Z 347.702,A -85,B 0,C 180,E1 -18649.973,E2 -18649.973} C_VEL
LIN {X 0,Y 264.232,Z 337.858,A -85,B 0,C 180,E1 -18651.862,E2 -18651.862} C_VEL
LIN {X 0,Y 266.261,Z 326.916,A -85,B 0,C 180,E1 -18653.509,E2 -18653.509} C_VEL
LIN {X 0,Y 266.24,Z 323.099,A -85,B 0,C 180,E1 -18654.066,E2 -18654.066} C_VEL
LIN {X 0,Y 264.573,Z 311.961,A -85,B 0,C 180,E1 -18655.621,E2 -18655.621} C_VEL
LIN {X 0,Y 262.144,Z 301.109,A -85,B 0,C 180,E1 -18656.949,E2 -18656.949} C_VEL
LIN {X 0,Y 258.673,Z 289.223,A -85,B 0,C 180,E1 -18658.219,E2 -18658.219} C_VEL
LIN {X 0,Y 255.827,Z 281.381,A -85,B 0,C 180,E1 -18658.984,E2 -18658.984} C_VEL
LIN {X 0,Y 255.703,Z 280.575,A -85,B 0,C 180,E1 -18659.073,E2 -18659.073} C_VEL
LIN {X 0,Y 255.95,Z 278.356,A -85,B 0,C 180,E1 -18661.656,E2 -18661.656} C_VEL
LIN {X 0,Y 256.214,Z 275.439,A -85,B 0,C 180,E1 -18665.172,E2 -18665.172} C_VEL
LIN {X 0,Y 256.262,Z 273.759,A -85,B 0,C 180,E1 -18667.314,E2 -18667.314} C_VEL
LIN {X 0,Y 256.098,Z 271.924,A -85,B 0,C 180,E1 -18669.79,E2 -18669.79} C_VEL
LIN {X 0,Y 256.032,Z 271.588,A -85,B 0,C 180,E1 -18672.171,E2 -18672.171} C_VEL
LIN {X 0,Y 256.051,Z 271.59,A -85,B 0,C 180,E1 -18676.67,E2 -18676.67} C_VEL
LIN {X 0,Y 256.074,Z 271.586,A -85,B 0,C 180,E1 -18680.858,E2 -18680.858} C_VEL
LIN {X 0,Y 256.118,Z 271.581,A -85,B 0,C 180,E1 -18684.812,E2 -18684.812} C_VEL
LIN {X 0,Y 256.095,Z 271.581,A -85,B 0,C 180,E1 -18688.573,E2 -18688.573} C_VEL
LIN {X 0,Y 256.144,Z 271.575,A -85,B 0,C 180,E1 -18692.196,E2 -18692.196} C_VEL
LIN {X 0,Y 256.145,Z 271.577,A -85,B 0,C 180,E1 -18695.697,E2 -18695.697} C_VEL
LIN {X 0,Y 256.151,Z 271.578,A -85,B 0,C 180,E1 -18699.103,E2 -18699.103} C_VEL
LIN {X 0,Y 256.261,Z 271.563,A -85,B 0,C 180,E1 -18704.082,E2 -18704.082} C_VEL
LIN {X 0,Y 256.29,Z 271.561,A -85,B 0,C 180,E1 -18707.327,E2 -18707.327} C_VEL
LIN {X 0,Y 256.498,Z 271.533,A -85,B 0,C 180,E1 -18712.126,E2 -18712.126} C_VEL
LIN {X 0,Y 256.46,Z 271.54,A -85,B 0,C 180,E1 -18716.858,E2 -18716.858} C_VEL
LIN {X 0,Y 256.7,Z 271.509,A -85,B 0,C 180,E1 -18718.431,E2 -18718.431} C_VEL
LIN {X 0,Y 256.716,Z 271.505,A -85,B 0,C 180,E1 -18721.569,E2 -18721.569} C_VEL
LIN {X 0,Y 256.477,Z 271.538,A -85,B 0,C 180,E1 -18726.293,E2 -18726.293} C_VEL
LIN {X 0,Y 256.429,Z 271.541,A -85,B 0,C 180,E1 -18729.465,E2 -18729.465} C_VEL
LIN {X 0,Y 256.257,Z 271.566,A -85,B 0,C 180,E1 -18734.29,E2 -18734.29} C_VEL
LIN {X 0,Y 256.214,Z 271.568,A -85,B 0,C 180,E1 -18737.562,E2 -18737.562} C_VEL
LIN {X 0,Y 256.154,Z 271.576,A -85,B 0,C 180,E1 -18741.116,E2 -18741.116} C_VEL
LIN {X 0,Y 256.107,Z 271.582,A -85,B 0,C 180,E1 -18745.098,E2 -18745.098} C_VEL
LIN {X 0,Y 256.056,Z 271.591,A -85,B 0,C 180,E1 -18749.53,E2 -18749.53} C_VEL
LIN {X 0,Y 255.402,Z 271.679,A -85,B 0,C 180,E1 -18750.843,E2 -18750.843} C_VEL
LIN {X 0,Y 252.579,Z 272.035,A -85,B 0,C 180,E1 -18752.983,E2 -18752.983} C_VEL
LIN {X 0,Y 250.165,Z 272.332,A -85,B 0,C 180,E1 -18754.725,E2 -18754.725} C_VEL
LIN {X 0,Y 249.114,Z 272.458,A -85,B 0,C 180,E1 -18756.075,E2 -18756.075} C_VEL
LIN {X 0,Y 249.021,Z 272.467,A -85,B 0,C 180,E1 -18756.533,E2 -18756.533} C_VEL
LIN {X 0,Y 249.015,Z 272.497,A -85,B 0,C 180,E1 -18759.889,E2 -18759.889} C_VEL
LIN {X 0,Y 249.418,Z 274.991,A -85,B 0,C 180,E1 -18762.893,E2 -18762.893} C_VEL
LIN {X 0,Y 250.082,Z 278.583,A -85,B 0,C 180,E1 -18766.943,E2 -18766.943} C_VEL
LIN {X 0,Y 250.507,Z 281.285,A -85,B 0,C 180,E1 -18769.814,E2 -18769.814} C_VEL
LIN {X 0,Y 250.783,Z 284.423,A -85,B 0,C 180,E1 -18772.949,E2 -18772.949} C_VEL
LIN {X 0,Y 250.445,Z 287.517,A -85,B 0,C 180,E1 -18775.858,E2 -18775.858} C_VEL
LIN {X 0,Y 249.444,Z 292.29,A -85,B 0,C 180,E1 -18780.17,E2 -18780.17} C_VEL
LIN {X 0,Y 251.177,Z 298.502,A -85,B 0,C 180,E1 -18780.707,E2 -18780.707} C_VEL
LIN {X 0,Y 254.193,Z 310.49,A -85,B 0,C 180,E1 -18781.881,E2 -18781.881} C_VEL
LIN {X 0,Y 256.278,Z 321.879,A -85,B 0,C 180,E1 -18783.175,E2 -18783.175} C_VEL
LIN {X 0,Y 257.541,Z 333.727,A -85,B 0,C 180,E1 -18784.733,E2 -18784.733} C_VEL
LIN {X 0,Y 257.95,Z 343.991,A -85,B 0,C 180,E1 -18786.304,E2 -18786.304} C_VEL
LIN {X 0,Y 255.931,Z 354.416,A -85,B 0,C 180,E1 -18788.028,E2 -18788.028} C_VEL
LIN {X 0,Y 253.978,Z 362.936,A -85,B 0,C 180,E1 -18789.763,E2 -18789.763} C_VEL
LIN {X 0,Y 252.391,Z 370.513,A -85,B 0,C 180,E1 -18791.66,E2 -18791.66} C_VEL
LIN {X 0,Y 250.53,Z 378.491,A -85,B 0,C 180,E1 -18794.126,E2 -18794.126} C_VEL
LIN {X 0,Y 248.776,Z 385.578,A -85,B 0,C 180,E1 -18796.938,E2 -18796.938} C_VEL
LIN {X 0,Y 247.849,Z 390.299,A -85,B 0,C 180,E1 -18799.379,E2 -18799.379} C_VEL
LIN {X 0,Y 247.264,Z 393.909,A -85,B 0,C 180,E1 -18801.83,E2 -18801.83} C_VEL
LIN {X 0,Y 247.009,Z 395.77,A -85,B 0,C 180,E1 -18803.465,E2 -18803.465} C_VEL
LIN {X 0,Y 246.883,Z 397.167,A -85,B 0,C 180,E1 -18805.101,E2 -18805.101} C_VEL
LIN {X 0,Y 246.865,Z 398.167,A -85,B 0,C 180,E1 -18806.736,E2 -18806.736} C_VEL
LIN {X 0,Y 246.928,Z 398.777,A -85,B 0,C 180,E1 -18808.369,E2 -18808.369} C_VEL
LIN {X 0,Y 246.984,Z 398.992,A -85,B 0,C 180,E1 -18810,E2 -18810} C_VEL
LIN {X 0,Y 246.927,Z 398.768,A -85,B 0,C 180,E1 -18811.631,E2 -18811.631} C_VEL
LIN {X 0,Y 246.883,Z 397.147,A -85,B 0,C 180,E1 -18814.899,E2 -18814.899} C_VEL
LIN {X 0,Y 246.982,Z 395.739,A -85,B 0,C 180,E1 -18816.536,E2 -18816.536} C_VEL
LIN {X 0,Y 247.418,Z 392.79,A -85,B 0,C 180,E1 -18818.988,E2 -18818.988} C_VEL
LIN {X 0,Y 248.14,Z 388.802,A -85,B 0,C 180,E1 -18821.435,E2 -18821.435} C_VEL
LIN {X 0,Y 249.439,Z 382.674,A -85,B 0,C 180,E1 -18824.272,E2 -18824.272} C_VEL
LIN {X 0,Y 251.09,Z 375.989,A -85,B 0,C 180,E1 -18826.672,E2 -18826.672} C_VEL
LIN {X 0,Y 252.937,Z 368.036,A -85,B 0,C 180,E1 -18828.959,E2 -18828.959} C_VEL
LIN {X 0,Y 254.825,Z 359.188,A -85,B 0,C 180,E1 -18831.01,E2 -18831.01} C_VEL
LIN {X 0,Y 257.106,Z 348.685,A -85,B 0,C 180,E1 -18832.925,E2 -18832.925} C_VEL
LIN {X 0,Y 257.89,Z 343.758,A -85,B 0,C 180,E1 -18833.701,E2 -18833.701} C_VEL
LIN {X 0,Y 257.455,Z 333.591,A -85,B 0,C 180,E1 -18835.255,E2 -18835.255} C_VEL
LIN {X 0,Y 256.408,Z 322.846,A -85,B 0,C 180,E1 -18836.663,E2 -18836.663} C_VEL
LIN {X 0,Y 254.277,Z 310.965,A -85,B 0,C 180,E1 -18838.026,E2 -18838.026} C_VEL
LIN {X 0,Y 251.081,Z 298.234,A -85,B 0,C 180,E1 -18839.274,E2 -18839.274} C_VEL
LIN {X 0,Y 249.444,Z 292.29,A -85,B 0,C 180,E1 -18839.788,E2 -18839.788} C_VEL
LIN {X 0,Y 250.442,Z 287.468,A -85,B 0,C 180,E1 -18844.142,E2 -18844.142} C_VEL
LIN {X 0,Y 250.772,Z 284.345,A -85,B 0,C 180,E1 -18847.053,E2 -18847.053} C_VEL
LIN {X 0,Y 250.408,Z 280.71,A -85,B 0,C 180,E1 -18850.73,E2 -18850.73} C_VEL
LIN {X 0,Y 249.8,Z 277.046,A -85,B 0,C 180,E1 -18854.697,E2 -18854.697} C_VEL
LIN {X 0,Y 249.107,Z 272.905,A -85,B 0,C 180,E1 -18859.542,E2 -18859.542} C_VEL
LIN {X 0,Y 249.012,Z 272.47,A -85,B 0,C 180,E1 -18860.123,E2 -18860.123} C_VEL
LIN {X 0,Y 249.027,Z 272.466,A -85,B 0,C 180,E1 -18863.654,E2 -18863.654} C_VEL
LIN {X 0,Y 249.034,Z 272.468,A -85,B 0,C 180,E1 -18867.847,E2 -18867.847} C_VEL
LIN {X 0,Y 249.049,Z 272.465,A -85,B 0,C 180,E1 -18871.332,E2 -18871.332} C_VEL
LIN {X 0,Y 249.077,Z 272.46,A -85,B 0,C 180,E1 -18874.96,E2 -18874.96} C_VEL
LIN {X 0,Y 249.089,Z 272.458,A -85,B 0,C 180,E1 -18878.605,E2 -18878.605} C_VEL
LIN {X 0,Y 249.243,Z 272.44,A -85,B 0,C 180,E1 -18883.622,E2 -18883.622} C_VEL
LIN {X 0,Y 249.244,Z 272.436,A -85,B 0,C 180,E1 -18888.616,E2 -18888.616} C_VEL
LIN {X 0,Y 249.447,Z 272.412,A -85,B 0,C 180,E1 -18891.902,E2 -18891.902} C_VEL
LIN {X 0,Y 249.295,Z 272.431,A -85,B 0,C 180,E1 -18895.149,E2 -18895.149} C_VEL
LIN {X 0,Y 249.677,Z 272.381,A -85,B 0,C 180,E1 -18898.387,E2 -18898.387} C_VEL
LIN {X 0,Y 249.664,Z 272.385,A -85,B 0,C 180,E1 -18901.613,E2 -18901.613} C_VEL
LIN {X 0,Y 249.43,Z 272.412,A -85,B 0,C 180,E1 -18906.705,E2 -18906.705} C_VEL
LIN {X 0,Y 249.344,Z 272.424,A -85,B 0,C 180,E1 -18909.737,E2 -18909.737} C_VEL
LIN {X 0,Y 249.184,Z 272.446,A -85,B 0,C 180,E1 -18914.705,E2 -18914.705} C_VEL
LIN {X 0,Y 249.113,Z 272.453,A -85,B 0,C 180,E1 -18918.079,E2 -18918.079} C_VEL
LIN {X 0,Y 249.082,Z 272.455,A -85,B 0,C 180,E1 -18921.519,E2 -18921.519} C_VEL
LIN {X 0,Y 249.119,Z 272.452,A -85,B 0,C 180,E1 -18925.476,E2 -18925.476} C_VEL
LIN {X 0,Y 249.088,Z 272.455,A -85,B 0,C 180,E1 -18928.995,E2 -18928.995} C_VEL
LIN {X 0,Y 249.035,Z 272.465,A -85,B 0,C 180,E1 -18932.425,E2 -18932.425} C_VEL
LIN {X 0,Y 249.065,Z 272.461,A -85,B 0,C 180,E1 -18936.34,E2 -18936.34} C_VEL
LIN {X 0,Y 249.007,Z 272.468,A -85,B 0,C 180,E1 -18940.478,E2 -18940.478} C_VEL
LIN {X 0,Y 248.984,Z 272.469,A -85,B 0,C 180,E1 -18944.884,E2 -18944.884} C_VEL
LIN {X 0,Y 248.984,Z 272.473,A -85,B 0,C 180,E1 -18947.356,E2 -18947.356} C_VEL
LIN {X 0,Y 248.998,Z 272.601,A -85,B 0,C 180,E1 -18949.648,E2 -18949.648} C_VEL
LIN {X 0,Y 249.213,Z 274.397,A -85,B 0,C 180,E1 -18952.151,E2 -18952.151} C_VEL
LIN {X 0,Y 249.171,Z 277.067,A -85,B 0,C 180,E1 -18955.659,E2 -18955.659} C_VEL
LIN {X 0,Y 248.806,Z 280.184,A -85,B 0,C 180,E1 -18959.44,E2 -18959.44} C_VEL
LIN {X 0,Y 248.746,Z 280.805,A -85,B 0,C 180,E1 -18960.182,E2 -18960.182} C_VEL
LIN {X 0,Y 250.702,Z 286.555,A -85,B 0,C 180,E1 -18960.756,E2 -18960.756} C_VEL
LIN {X 0,Y 254.42,Z 297.79,A -85,B 0,C 180,E1 -18961.992,E2 -18961.992} C_VEL
LIN {X 0,Y 257.294,Z 309.79,A -85,B 0,C 180,E1 -18963.467,E2 -18963.467} C_VEL
LIN {X 0,Y 259.103,Z 320.658,A -85,B 0,C 180,E1 -18964.992,E2 -18964.992} C_VEL
LIN {X 0,Y 259.71,Z 326.419,A -85,B 0,C 180,E1 -18965.886,E2 -18965.886} C_VEL
LIN {X 0,Y 257.763,Z 337.398,A -85,B 0,C 180,E1 -18967.56,E2 -18967.56} C_VEL
LIN {X 0,Y 255.685,Z 347.361,A -85,B 0,C 180,E1 -18969.485,E2 -18969.485} C_VEL
LIN {X 0,Y 253.508,Z 356.996,A -85,B 0,C 180,E1 -18971.827,E2 -18971.827} C_VEL
LIN {X 0,Y 251.499,Z 364.681,A -85,B 0,C 180,E1 -18974.19,E2 -18974.19} C_VEL
LIN {X 0,Y 250.213,Z 369.924,A -85,B 0,C 180,E1 -18976.187,E2 -18976.187} C_VEL
LIN {X 0,Y 248.965,Z 375.009,A -85,B 0,C 180,E1 -18978.603,E2 -18978.603} C_VEL
LIN {X 0,Y 248.071,Z 378.955,A -85,B 0,C 180,E1 -18981.036,E2 -18981.036} C_VEL
LIN {X 0,Y 247.394,Z 382.23,A -85,B 0,C 180,E1 -18983.874,E2 -18983.874} C_VEL
LIN {X 0,Y 247.095,Z 384.25,A -85,B 0,C 180,E1 -18986.739,E2 -18986.739} C_VEL
LIN {X 0,Y 246.993,Z 385.088,A -85,B 0,C 180,E1 -18990,E2 -18990} C_VEL
LIN {X 0,Y 247.004,Z 384.895,A -85,B 0,C 180,E1 -18991.631,E2 -18991.631} C_VEL
LIN {X 0,Y 247.094,Z 384.309,A -85,B 0,C 180,E1 -18993.261,E2 -18993.261} C_VEL
LIN {X 0,Y 247.503,Z 381.985,A -85,B 0,C 180,E1 -18996.522,E2 -18996.522} C_VEL
LIN {X 0,Y 248.102,Z 379.118,A -85,B 0,C 180,E1 -18998.963,E2 -18998.963} C_VEL
LIN {X 0,Y 248.944,Z 375.229,A -85,B 0,C 180,E1 -19001.398,E2 -19001.398} C_VEL
LIN {X 0,Y 250.192,Z 370.209,A -85,B 0,C 180,E1 -19003.814,E2 -19003.814} C_VEL
LIN {X 0,Y 251.739,Z 363.886,A -85,B 0,C 180,E1 -19006.211,E2 -19006.211} C_VEL
LIN {X 0,Y 253.756,Z 355.97,A -85,B 0,C 180,E1 -19008.573,E2 -19008.573} C_VEL
LIN {X 0,Y 255.652,Z 347.944,A -85,B 0,C 180,E1 -19010.508,E2 -19010.508} C_VEL
LIN {X 0,Y 257.64,Z 338.054,A -85,B 0,C 180,E1 -19012.451,E2 -19012.451} C_VEL
LIN {X 0,Y 259.739,Z 327.209,A -85,B 0,C 180,E1 -19014.121,E2 -19014.121} C_VEL
LIN {X 0,Y 258.669,Z 317.388,A -85,B 0,C 180,E1 -19015.618,E2 -19015.618} C_VEL
LIN {X 0,Y 256.569,Z 306.456,A -85,B 0,C 180,E1 -19017.097,E2 -19017.097} C_VEL
LIN {X 0,Y 253.471,Z 294.582,A -85,B 0,C 180,E1 -19018.501,E2 -19018.501} C_VEL
LIN {X 0,Y 249.508,Z 283.485,A -85,B 0,C 180,E1 -19019.694,E2 -19019.694} C_VEL
LIN {X 0,Y 248.734,Z 280.795,A -85,B 0,C 180,E1 -19019.973,E2 -19019.973} C_VEL
LIN {X 0,Y 249.129,Z 277.184,A -85,B 0,C 180,E1 -19024.348,E2 -19024.348} C_VEL
LIN {X 0,Y 249.164,Z 274.137,A -85,B 0,C 180,E1 -19028.356,E2 -19028.356} C_VEL
LIN {X 0,Y 248.99,Z 272.613,A -85,B 0,C 180,E1 -19030.482,E2 -19030.482} C_VEL
LIN {X 0,Y 248.985,Z 272.468,A -85,B 0,C 180,E1 -19034.884,E2 -19034.884} C_VEL
LIN {X 0,Y 249.011,Z 272.466,A -85,B 0,C 180,E1 -19037.361,E2 -19037.361} C_VEL
LIN {X 0,Y 249.03,Z 272.464,A -85,B 0,C 180,E1 -19041.62,E2 -19041.62} C_VEL
LIN {X 0,Y 249.061,Z 272.461,A -85,B 0,C 180,E1 -19045.642,E2 -19045.642} C_VEL
LIN {X 0,Y 249.055,Z 272.459,A -85,B 0,C 180,E1 -19049.473,E2 -19049.473} C_VEL
LIN {X 0,Y 249.073,Z 272.456,A -85,B 0,C 180,E1 -19053.162,E2 -19053.162} C_VEL
LIN {X 0,Y 249.063,Z 272.455,A -85,B 0,C 180,E1 -19056.731,E2 -19056.731} C_VEL
LIN {X 0,Y 249.088,Z 272.456,A -85,B 0,C 180,E1 -19060.21,E2 -19060.21} C_VEL
LIN {X 0,Y 249.198,Z 272.445,A -85,B 0,C 180,E1 -19063.619,E2 -19063.619} C_VEL
LIN {X 0,Y 249.244,Z 272.436,A -85,B 0,C 180,E1 -19068.616,E2 -19068.616} C_VEL
LIN {X 0,Y 249.442,Z 272.412,A -85,B 0,C 180,E1 -19071.901,E2 -19071.901} C_VEL
LIN {X 0,Y 249.275,Z 272.435,A -85,B 0,C 180,E1 -19075.148,E2 -19075.148} C_VEL
LIN {X 0,Y 249.662,Z 272.386,A -85,B 0,C 180,E1 -19078.387,E2 -19078.387} C_VEL
LIN {X 0,Y 249.677,Z 272.382,A -85,B 0,C 180,E1 -19081.613,E2 -19081.613} C_VEL
LIN {X 0,Y 249.449,Z 272.415,A -85,B 0,C 180,E1 -19086.471,E2 -19086.471} C_VEL
LIN {X 0,Y 249.346,Z 272.424,A -85,B 0,C 180,E1 -19089.736,E2 -19089.736} C_VEL
LIN {X 0,Y 249.208,Z 272.442,A -85,B 0,C 180,E1 -19094.703,E2 -19094.703} C_VEL
LIN {X 0,Y 249.142,Z 272.452,A -85,B 0,C 180,E1 -19098.077,E2 -19098.077} C_VEL
LIN {X 0,Y 249.085,Z 272.457,A -85,B 0,C 180,E1 -19101.518,E2 -19101.518} C_VEL
LIN {X 0,Y 249.064,Z 272.46,A -85,B 0,C 180,E1 -19105.449,E2 -19105.449} C_VEL
LIN {X 0,Y 249.005,Z 272.465,A -85,B 0,C 180,E1 -19109.516,E2 -19109.516} C_VEL
LIN {X 0,Y 249.029,Z 272.466,A -85,B 0,C 180,E1 -19112.426,E2 -19112.426} C_VEL
LIN {X 0,Y 249.021,Z 272.467,A -85,B 0,C 180,E1 -19116.533,E2 -19116.533} C_VEL
LIN {X 0,Y 248.354,Z 272.711,A -85,B 0,C 180,E1 -19117.882,E2 -19117.882} C_VEL
LIN {X 0,Y 245.637,Z 273.939,A -85,B 0,C 180,E1 -19120.075,E2 -19120.075} C_VEL
LIN {X 0,Y 243.417,Z 275.38,A -85,B 0,C 180,E1 -19121.848,E2 -19121.848} C_VEL
LIN {X 0,Y 242.57,Z 276.567,A -85,B 0,C 180,E1 -19123.215,E2 -19123.215} C_VEL
LIN {X 0,Y 242.555,Z 276.962,A -85,B 0,C 180,E1 -19123.676,E2 -19123.676} C_VEL
LIN {X 0,Y 242.977,Z 279.239,A -85,B 0,C 180,E1 -19126.312,E2 -19126.312} C_VEL
LIN {X 0,Y 243.571,Z 283.162,A -85,B 0,C 180,E1 -19130.595,E2 -19130.595} C_VEL
LIN {X 0,Y 243.697,Z 286.375,A -85,B 0,C 180,E1 -19133.852,E2 -19133.852} C_VEL
LIN {X 0,Y 243.111,Z 289.637,A -85,B 0,C 180,E1 -19136.966,E2 -19136.966} C_VEL
LIN {X 0,Y 242.576,Z 292.113,A -85,B 0,C 180,E1 -19139.253,E2 -19139.253} C_VEL
LIN {X 0,Y 243.466,Z 295.378,A -85,B 0,C 180,E1 -19139.532,E2 -19139.532} C_VEL
LIN {X 0,Y 246.883,Z 307.996,A -85,B 0,C 180,E1 -19140.794,E2 -19140.794} C_VEL
LIN {X 0,Y 249.302,Z 320.041,A -85,B 0,C 180,E1 -19142.188,E2 -19142.188} C_VEL
LIN {X 0,Y 250.572,Z 330.464,A -85,B 0,C 180,E1 -19143.561,E2 -19143.561} C_VEL
LIN {X 0,Y 251.178,Z 341.169,A -85,B 0,C 180,E1 -19145.184,E2 -19145.184} C_VEL
LIN {X 0,Y 251.076,Z 346.346,A -85,B 0,C 180,E1 -19146.054,E2 -19146.054} C_VEL
LIN {X 0,Y 248.614,Z 357.211,A -85,B 0,C 180,E1 -19148.003,E2 -19148.003} C_VEL
LIN {X 0,Y 246.496,Z 366.043,A -85,B 0,C 180,E1 -19149.992,E2 -19149.992} C_VEL
LIN {X 0,Y 244.861,Z 373.342,A -85,B 0,C 180,E1 -19152.028,E2 -19152.028} C_VEL
LIN {X 0,Y 243.073,Z 380.528,A -85,B 0,C 180,E1 -19154.487,E2 -19154.487} C_VEL
LIN {X 0,Y 241.822,Z 385.379,A -85,B 0,C 180,E1 -19156.555,E2 -19156.555} C_VEL
LIN {X 0,Y 240.851,Z 390.1,A -85,B 0,C 180,E1 -19159.066,E2 -19159.066} C_VEL
LIN {X 0,Y 240.211,Z 393.709,A -85,B 0,C 180,E1 -19161.588,E2 -19161.588} C_VEL
LIN {X 0,Y 239.926,Z 395.57,A -85,B 0,C 180,E1 -19163.271,E2 -19163.271} C_VEL
LIN {X 0,Y 239.793,Z 397.135,A -85,B 0,C 180,E1 -19165.202,E2 -19165.202} C_VEL
LIN {X 0,Y 239.838,Z 398.578,A -85,B 0,C 180,E1 -19168.321,E2 -19168.321} C_VEL
LIN {X 0,Y 239.893,Z 398.792,A -85,B 0,C 180,E1 -19170,E2 -19170} C_VEL
LIN {X 0,Y 239.836,Z 398.568,A -85,B 0,C 180,E1 -19171.679,E2 -19171.679} C_VEL
LIN {X 0,Y 239.8,Z 396.946,A -85,B 0,C 180,E1 -19175.044,E2 -19175.044} C_VEL
LIN {X 0,Y 239.908,Z 395.538,A -85,B 0,C 180,E1 -19176.729,E2 -19176.729} C_VEL
LIN {X 0,Y 240.383,Z 392.588,A -85,B 0,C 180,E1 -19179.253,E2 -19179.253} C_VEL
LIN {X 0,Y 241.161,Z 388.6,A -85,B 0,C 180,E1 -19181.771,E2 -19181.771} C_VEL
LIN {X 0,Y 242.547,Z 382.472,A -85,B 0,C 180,E1 -19184.687,E2 -19184.687} C_VEL
LIN {X 0,Y 244.231,Z 375.785,A -85,B 0,C 180,E1 -19187.155,E2 -19187.155} C_VEL
LIN {X 0,Y 246.375,Z 367.006,A -85,B 0,C 180,E1 -19189.721,E2 -19189.721} C_VEL
LIN {X 0,Y 248.189,Z 358.985,A -85,B 0,C 180,E1 -19191.6,E2 -19191.6} C_VEL
LIN {X 0,Y 250.566,Z 348.482,A -85,B 0,C 180,E1 -19193.559,E2 -19193.559} C_VEL
LIN {X 0,Y 251.168,Z 344.849,A -85,B 0,C 180,E1 -19194.156,E2 -19194.156} C_VEL
LIN {X 0,Y 250.815,Z 334.461,A -85,B 0,C 180,E1 -19195.822,E2 -19195.822} C_VEL
LIN {X 0,Y 249.804,Z 323.798,A -85,B 0,C 180,E1 -19197.294,E2 -19197.294} C_VEL
LIN {X 0,Y 247.785,Z 311.994,A -85,B 0,C 180,E1 -19198.717,E2 -19198.717} C_VEL
LIN {X 0,Y 244.61,Z 299.296,A -85,B 0,C 180,E1 -19200.056,E2 -19200.056} C_VEL
LIN {X 0,Y 242.633,Z 292.658,A -85,B 0,C 180,E1 -19200.668,E2 -19200.668} C_VEL
LIN {X 0,Y 242.57,Z 292.01,A -85,B 0,C 180,E1 -19200.778,E2 -19200.778} C_VEL
LIN {X 0,Y 243.422,Z 288.281,A -85,B 0,C 180,E1 -19204.263,E2 -19204.263} C_VEL
LIN {X 0,Y 243.744,Z 285.179,A -85,B 0,C 180,E1 -19207.265,E2 -19207.265} C_VEL
LIN {X 0,Y 243.576,Z 283.101,A -85,B 0,C 180,E1 -19209.403,E2 -19209.403} C_VEL
LIN {X 0,Y 242.965,Z 279.167,A -85,B 0,C 180,E1 -19213.685,E2 -19213.685} C_VEL
LIN {X 0,Y 242.289,Z 275.393,A -85,B 0,C 180,E1 -19218.152,E2 -19218.152} C_VEL
LIN {X 0,Y 241.988,Z 273.344,A -85,B 0,C 180,E1 -19220.852,E2 -19220.852} C_VEL
LIN {X 0,Y 241.98,Z 273.346,A -85,B 0,C 180,E1 -19224.488,E2 -19224.488} C_VEL
LIN {X 0,Y 241.954,Z 273.352,A -85,B 0,C 180,E1 -19228.477,E2 -19228.477} C_VEL
LIN {X 0,Y 241.964,Z 273.349,A -85,B 0,C 180,E1 -19232.307,E2 -19232.307} C_VEL
LIN {X 0,Y 242.01,Z 273.342,A -85,B 0,C 180,E1 -19236.011,E2 -19236.011} C_VEL
LIN {X 0,Y 242.03,Z 273.338,A -85,B 0,C 180,E1 -19239.607,E2 -19239.607} C_VEL
LIN {X 0,Y 242.164,Z 273.32,A -85,B 0,C 180,E1 -19243.278,E2 -19243.278} C_VEL
LIN {X 0,Y 242.181,Z 273.317,A -85,B 0,C 180,E1 -19248.28,E2 -19248.28} C_VEL
LIN {X 0,Y 242.395,Z 273.291,A -85,B 0,C 180,E1 -19251.665,E2 -19251.665} C_VEL
LIN {X 0,Y 242.255,Z 273.308,A -85,B 0,C 180,E1 -19255.007,E2 -19255.007} C_VEL
LIN {X 0,Y 242.637,Z 273.257,A -85,B 0,C 180,E1 -19258.34,E2 -19258.34} C_VEL
LIN {X 0,Y 242.623,Z 273.261,A -85,B 0,C 180,E1 -19261.66,E2 -19261.66} C_VEL
LIN {X 0,Y 242.411,Z 273.289,A -85,B 0,C 180,E1 -19266.677,E2 -19266.677} C_VEL
LIN {X 0,Y 242.267,Z 273.306,A -85,B 0,C 180,E1 -19270.024,E2 -19270.024} C_VEL
LIN {X 0,Y 242.14,Z 273.322,A -85,B 0,C 180,E1 -19275.143,E2 -19275.143} C_VEL
LIN {X 0,Y 242.051,Z 273.334,A -85,B 0,C 180,E1 -19278.626,E2 -19278.626} C_VEL
LIN {X 0,Y 242.006,Z 273.339,A -85,B 0,C 180,E1 -19282.181,E2 -19282.181} C_VEL
LIN {X 0,Y 242.068,Z 273.332,A -85,B 0,C 180,E1 -19285.838,E2 -19285.838} C_VEL
LIN {X 0,Y 242.033,Z 273.334,A -85,B 0,C 180,E1 -19289.58,E2 -19289.58} C_VEL
LIN {X 0,Y 241.99,Z 273.341,A -85,B 0,C 180,E1 -19293.491,E2 -19293.491} C_VEL
LIN {X 0,Y 241.996,Z 273.341,A -85,B 0,C 180,E1 -19297.581,E2 -19297.581} C_VEL
LIN {X 0,Y 241.935,Z 273.348,A -85,B 0,C 180,E1 -19301.923,E2 -19301.923} C_VEL
LIN {X 0,Y 241.909,Z 273.351,A -85,B 0,C 180,E1 -19306.578,E2 -19306.578} C_VEL
LIN {X 0,Y 241.917,Z 273.393,A -85,B 0,C 180,E1 -19309.055,E2 -19309.055} C_VEL
LIN {X 0,Y 242.207,Z 275.753,A -85,B 0,C 180,E1 -19312.458,E2 -19312.458} C_VEL
LIN {X 0,Y 242.196,Z 277.281,A -85,B 0,C 180,E1 -19314.525,E2 -19314.525} C_VEL
LIN {X 0,Y 241.865,Z 280.387,A -85,B 0,C 180,E1 -19318.464,E2 -19318.464} C_VEL
LIN {X 0,Y 241.808,Z 281.125,A -85,B 0,C 180,E1 -19319.269,E2 -19319.269} C_VEL
LIN {X 0,Y 243.823,Z 286.892,A -85,B 0,C 180,E1 -19319.852,E2 -19319.852} C_VEL
LIN {X 0,Y 247.616,Z 298.018,A -85,B 0,C 180,E1 -19321.151,E2 -19321.151} C_VEL
LIN {X 0,Y 250.521,Z 310.01,A -85,B 0,C 180,E1 -19322.691,E2 -19322.691} C_VEL
LIN {X 0,Y 252.274,Z 320.273,A -85,B 0,C 180,E1 -19324.182,E2 -19324.182} C_VEL
LIN {X 0,Y 253.07,Z 327.733,A -85,B 0,C 180,E1 -19325.382,E2 -19325.382} C_VEL
LIN {X 0,Y 251.216,Z 337.601,A -85,B 0,C 180,E1 -19326.942,E2 -19326.942} C_VEL
LIN {X 0,Y 249.2,Z 346.739,A -85,B 0,C 180,E1 -19328.724,E2 -19328.724} C_VEL
LIN {X 0,Y 247.117,Z 355.72,A -85,B 0,C 180,E1 -19330.91,E2 -19330.91} C_VEL
LIN {X 0,Y 244.991,Z 363.714,A -85,B 0,C 180,E1 -19333.33,E2 -19333.33} C_VEL
LIN {X 0,Y 243.323,Z 370.126,A -85,B 0,C 180,E1 -19335.788,E2 -19335.788} C_VEL
LIN {X 0,Y 242.001,Z 375.21,A -85,B 0,C 180,E1 -19338.271,E2 -19338.271} C_VEL
LIN {X 0,Y 241.06,Z 379.155,A -85,B 0,C 180,E1 -19340.773,E2 -19340.773} C_VEL
LIN {X 0,Y 240.277,Z 382.68,A -85,B 0,C 180,E1 -19343.983,E2 -19343.983} C_VEL
LIN {X 0,Y 240.019,Z 384.449,A -85,B 0,C 180,E1 -19346.643,E2 -19346.643} C_VEL
LIN {X 0,Y 239.924,Z 385.286,A -85,B 0,C 180,E1 -19350,E2 -19350} C_VEL
LIN {X 0,Y 239.917,Z 385.094,A -85,B 0,C 180,E1 -19351.679,E2 -19351.679} C_VEL
LIN {X 0,Y 240.018,Z 384.508,A -85,B 0,C 180,E1 -19353.357,E2 -19353.357} C_VEL
LIN {X 0,Y 240.453,Z 382.184,A -85,B 0,C 180,E1 -19356.714,E2 -19356.714} C_VEL
LIN {X 0,Y 241.097,Z 379.316,A -85,B 0,C 180,E1 -19359.226,E2 -19359.226} C_VEL
LIN {X 0,Y 241.975,Z 375.428,A -85,B 0,C 180,E1 -19361.731,E2 -19361.731} C_VEL
LIN {X 0,Y 243.293,Z 370.407,A -85,B 0,C 180,E1 -19364.214,E2 -19364.214} C_VEL
LIN {X 0,Y 244.935,Z 364.084,A -85,B 0,C 180,E1 -19366.675,E2 -19366.675} C_VEL
LIN {X 0,Y 247.041,Z 356.167,A -85,B 0,C 180,E1 -19369.097,E2 -19369.097} C_VEL
LIN {X 0,Y 249.087,Z 347.656,A -85,B 0,C 180,E1 -19371.192,E2 -19371.192} C_VEL
LIN {X 0,Y 251.087,Z 338.251,A -85,B 0,C 180,E1 -19373.071,E2 -19373.071} C_VEL
LIN {X 0,Y 253.134,Z 327.51,A -85,B 0,C 180,E1 -19374.777,E2 -19374.777} C_VEL
LIN {X 0,Y 251.752,Z 316.387,A -85,B 0,C 180,E1 -19376.53,E2 -19376.53} C_VEL
LIN {X 0,Y 249.19,Z 304,A -85,B 0,C 180,E1 -19378.241,E2 -19378.241} C_VEL
LIN {X 0,Y 245.797,Z 292.301,A -85,B 0,C 180,E1 -19379.668,E2 -19379.668} C_VEL
LIN {X 0,Y 241.86,Z 281.675,A -85,B 0,C 180,E1 -19380.84,E2 -19380.84} C_VEL
LIN {X 0,Y 241.775,Z 280.997,A -85,B 0,C 180,E1 -19380.935,E2 -19380.935} C_VEL
LIN {X 0,Y 241.995,Z 278.946,A -85,B 0,C 180,E1 -19383.491,E2 -19383.491} C_VEL
LIN {X 0,Y 242.181,Z 277.263,A -85,B 0,C 180,E1 -19385.654,E2 -19385.654} C_VEL
LIN {X 0,Y 242.158,Z 275.243,A -85,B 0,C 180,E1 -19388.408,E2 -19388.408} C_VEL
LIN {X 0,Y 241.918,Z 273.494,A -85,B 0,C 180,E1 -19390.945,E2 -19390.945} C_VEL
LIN {X 0,Y 241.912,Z 273.348,A -85,B 0,C 180,E1 -19394.207,E2 -19394.207} C_VEL
LIN {X 0,Y 241.936,Z 273.349,A -85,B 0,C 180,E1 -19398.077,E2 -19398.077} C_VEL
LIN {X 0,Y 241.998,Z 273.341,A -85,B 0,C 180,E1 -19402.419,E2 -19402.419} C_VEL
LIN {X 0,Y 241.991,Z 273.341,A -85,B 0,C 180,E1 -19406.509,E2 -19406.509} C_VEL
LIN {X 0,Y 242.04,Z 273.335,A -85,B 0,C 180,E1 -19410.587,E2 -19410.587} C_VEL
LIN {X 0,Y 242.07,Z 273.332,A -85,B 0,C 180,E1 -19414.183,E2 -19414.183} C_VEL
LIN {X 0,Y 242.026,Z 273.336,A -85,B 0,C 180,E1 -19418.315,E2 -19418.315} C_VEL
LIN {X 0,Y 242.13,Z 273.325,A -85,B 0,C 180,E1 -19423.307,E2 -19423.307} C_VEL
LIN {X 0,Y 242.18,Z 273.316,A -85,B 0,C 180,E1 -19428.279,E2 -19428.279} C_VEL
LIN {X 0,Y 242.391,Z 273.291,A -85,B 0,C 180,E1 -19431.664,E2 -19431.664} C_VEL
LIN {X 0,Y 242.236,Z 273.313,A -85,B 0,C 180,E1 -19435.007,E2 -19435.007} C_VEL
LIN {X 0,Y 242.622,Z 273.263,A -85,B 0,C 180,E1 -19438.34,E2 -19438.34} C_VEL
LIN {X 0,Y 242.638,Z 273.259,A -85,B 0,C 180,E1 -19441.66,E2 -19441.66} C_VEL
LIN {X 0,Y 242.42,Z 273.289,A -85,B 0,C 180,E1 -19446.659,E2 -19446.659} C_VEL
LIN {X 0,Y 242.27,Z 273.307,A -85,B 0,C 180,E1 -19450.024,E2 -19450.024} C_VEL
LIN {X 0,Y 242.169,Z 273.317,A -85,B 0,C 180,E1 -19455.141,E2 -19455.141} C_VEL
LIN {X 0,Y 242.075,Z 273.33,A -85,B 0,C 180,E1 -19458.624,E2 -19458.624} C_VEL
LIN {X 0,Y 242.003,Z 273.342,A -85,B 0,C 180,E1 -19462.181,E2 -19462.181} C_VEL
LIN {X 0,Y 241.995,Z 273.339,A -85,B 0,C 180,E1 -19465.825,E2 -19465.825} C_VEL
LIN {X 0,Y 241.97,Z 273.346,A -85,B 0,C 180,E1 -19469.588,E2 -19469.588} C_VEL
LIN {X 0,Y 241.981,Z 273.346,A -85,B 0,C 180,E1 -19473.493,E2 -19473.493} C_VEL
LIN {X 0,Y 241.985,Z 273.346,A -85,B 0,C 180,E1 -19477.583,E2 -19477.583} C_VEL
LIN {X 0,Y 241.996,Z 273.446,A -85,B 0,C 180,E1 -19479.334,E2 -19479.334} C_VEL
LIN {X 0,Y 242.555,Z 276.962,A -85,B 0,C 180,E1 -19483.676,E2 -19483.676} C_VEL
LIN {X 0,Y 242.108,Z 278.242,A -85,B 0,C 180,E1 -19485.033,E2 -19485.033} C_VEL
LIN {X 0,Y 239.637,Z 280.668,A -85,B 0,C 180,E1 -19487.242,E2 -19487.242} C_VEL
LIN {X 0,Y 237.494,Z 282.675,A -85,B 0,C 180,E1 -19489.036,E2 -19489.036} C_VEL
LIN {X 0,Y 236.63,Z 284.105,A -85,B 0,C 180,E1 -19490.425,E2 -19490.425} C_VEL
LIN {X 0,Y 236.594,Z 284.553,A -85,B 0,C 180,E1 -19490.896,E2 -19490.896} C_VEL
LIN {X 0,Y 236.683,Z 287.096,A -85,B 0,C 180,E1 -19493.567,E2 -19493.567} C_VEL
LIN {X 0,Y 236.183,Z 289.99,A -85,B 0,C 180,E1 -19496.428,E2 -19496.428} C_VEL
LIN {X 0,Y 235.788,Z 292.023,A -85,B 0,C 180,E1 -19498.271,E2 -19498.271} C_VEL
LIN {X 0,Y 237.619,Z 298.402,A -85,B 0,C 180,E1 -19498.873,E2 -19498.873} C_VEL
LIN {X 0,Y 240.646,Z 309.932,A -85,B 0,C 180,E1 -19500.131,E2 -19500.131} C_VEL
LIN {X 0,Y 242.965,Z 322.375,A -85,B 0,C 180,E1 -19501.683,E2 -19501.683} C_VEL
LIN {X 0,Y 244.097,Z 333.051,A -85,B 0,C 180,E1 -19503.195,E2 -19503.195} C_VEL
LIN {X 0,Y 244.499,Z 343.584,A -85,B 0,C 180,E1 -19504.914,E2 -19504.914} C_VEL
LIN {X 0,Y 244.338,Z 347.327,A -85,B 0,C 180,E1 -19505.576,E2 -19505.576} C_VEL
LIN {X 0,Y 242.046,Z 357.014,A -85,B 0,C 180,E1 -19507.373,E2 -19507.373} C_VEL
LIN {X 0,Y 239.807,Z 365.845,A -85,B 0,C 180,E1 -19509.409,E2 -19509.409} C_VEL
LIN {X 0,Y 238.105,Z 373.144,A -85,B 0,C 180,E1 -19511.5,E2 -19511.5} C_VEL
LIN {X 0,Y 236.222,Z 380.329,A -85,B 0,C 180,E1 -19514.026,E2 -19514.026} C_VEL
LIN {X 0,Y 234.883,Z 385.179,A -85,B 0,C 180,E1 -19516.15,E2 -19516.15} C_VEL
LIN {X 0,Y 233.869,Z 389.901,A -85,B 0,C 180,E1 -19518.736,E2 -19518.736} C_VEL
LIN {X 0,Y 233.178,Z 393.51,A -85,B 0,C 180,E1 -19521.332,E2 -19521.332} C_VEL
LIN {X 0,Y 232.872,Z 395.371,A -85,B 0,C 180,E1 -19523.066,E2 -19523.066} C_VEL
LIN {X 0,Y 232.692,Z 397.124,A -85,B 0,C 180,E1 -19525.344,E2 -19525.344} C_VEL
LIN {X 0,Y 232.749,Z 398.378,A -85,B 0,C 180,E1 -19528.269,E2 -19528.269} C_VEL
LIN {X 0,Y 232.803,Z 398.592,A -85,B 0,C 180,E1 -19530,E2 -19530} C_VEL
LIN {X 0,Y 232.747,Z 398.368,A -85,B 0,C 180,E1 -19531.73,E2 -19531.73} C_VEL
LIN {X 0,Y 232.729,Z 396.746,A -85,B 0,C 180,E1 -19535.198,E2 -19535.198} C_VEL
LIN {X 0,Y 232.83,Z 395.336,A -85,B 0,C 180,E1 -19536.935,E2 -19536.935} C_VEL
LIN {X 0,Y 233.367,Z 392.387,A -85,B 0,C 180,E1 -19539.534,E2 -19539.534} C_VEL
LIN {X 0,Y 234.174,Z 388.398,A -85,B 0,C 180,E1 -19542.127,E2 -19542.127} C_VEL
LIN {X 0,Y 235.663,Z 382.27,A -85,B 0,C 180,E1 -19545.126,E2 -19545.126} C_VEL
LIN {X 0,Y 237.407,Z 375.582,A -85,B 0,C 180,E1 -19547.664,E2 -19547.664} C_VEL
LIN {X 0,Y 239.478,Z 367.535,A -85,B 0,C 180,E1 -19550.097,E2 -19550.097} C_VEL
LIN {X 0,Y 241.594,Z 358.782,A -85,B 0,C 180,E1 -19552.22,E2 -19552.22} C_VEL
LIN {X 0,Y 244.052,Z 348.277,A -85,B 0,C 180,E1 -19554.227,E2 -19554.227} C_VEL
LIN {X 0,Y 244.469,Z 344.638,A -85,B 0,C 180,E1 -19554.862,E2 -19554.862} C_VEL
LIN {X 0,Y 244.041,Z 332.967,A -85,B 0,C 180,E1 -19556.778,E2 -19556.778} C_VEL
LIN {X 0,Y 242.937,Z 322.298,A -85,B 0,C 180,E1 -19558.282,E2 -19558.282} C_VEL
LIN {X 0,Y 240.77,Z 310.514,A -85,B 0,C 180,E1 -19559.751,E2 -19559.751} C_VEL
LIN {X 0,Y 237.529,Z 298.189,A -85,B 0,C 180,E1 -19561.1,E2 -19561.1} C_VEL
LIN {X 0,Y 235.753,Z 291.861,A -85,B 0,C 180,E1 -19561.72,E2 -19561.72} C_VEL
LIN {X 0,Y 236.548,Z 288.071,A -85,B 0,C 180,E1 -19565.405,E2 -19565.405} C_VEL
LIN {X 0,Y 236.644,Z 284.966,A -85,B 0,C 180,E1 -19568.585,E2 -19568.585} C_VEL
LIN {X 0,Y 236.194,Z 281.896,A -85,B 0,C 180,E1 -19571.937,E2 -19571.937} C_VEL
LIN {X 0,Y 235.628,Z 278.694,A -85,B 0,C 180,E1 -19575.712,E2 -19575.712} C_VEL
LIN {X 0,Y 235.243,Z 276.121,A -85,B 0,C 180,E1 -19578.909,E2 -19578.909} C_VEL
LIN {X 0,Y 234.953,Z 274.22,A -85,B 0,C 180,E1 -19581.634,E2 -19581.634} C_VEL
LIN {X 0,Y 234.926,Z 274.223,A -85,B 0,C 180,E1 -19585.361,E2 -19585.361} C_VEL
LIN {X 0,Y 234.899,Z 274.228,A -85,B 0,C 180,E1 -19589.428,E2 -19589.428} C_VEL
LIN {X 0,Y 234.946,Z 274.224,A -85,B 0,C 180,E1 -19593.818,E2 -19593.818} C_VEL
LIN {X 0,Y 234.993,Z 274.213,A -85,B 0,C 180,E1 -19598.968,E2 -19598.968} C_VEL
LIN {X 0,Y 235.097,Z 274.2,A -85,B 0,C 180,E1 -19603.06,E2 -19603.06} C_VEL
LIN {X 0,Y 235.115,Z 274.198,A -85,B 0,C 180,E1 -19607.922,E2 -19607.922} C_VEL
LIN {X 0,Y 235.327,Z 274.172,A -85,B 0,C 180,E1 -19611.412,E2 -19611.412} C_VEL
LIN {X 0,Y 235.369,Z 274.166,A -85,B 0,C 180,E1 -19613.14,E2 -19613.14} C_VEL
LIN {X 0,Y 235.597,Z 274.134,A -85,B 0,C 180,E1 -19618.291,E2 -19618.291} C_VEL
LIN {X 0,Y 235.582,Z 274.138,A -85,B 0,C 180,E1 -19621.71,E2 -19621.71} C_VEL
LIN {X 0,Y 235.364,Z 274.168,A -85,B 0,C 180,E1 -19626.86,E2 -19626.86} C_VEL
LIN {X 0,Y 235.213,Z 274.185,A -85,B 0,C 180,E1 -19630.328,E2 -19630.328} C_VEL
LIN {X 0,Y 235.087,Z 274.199,A -85,B 0,C 180,E1 -19635.608,E2 -19635.608} C_VEL
LIN {X 0,Y 234.991,Z 274.213,A -85,B 0,C 180,E1 -19639.207,E2 -19639.207} C_VEL
LIN {X 0,Y 234.953,Z 274.218,A -85,B 0,C 180,E1 -19642.884,E2 -19642.884} C_VEL
LIN {X 0,Y 234.972,Z 274.216,A -85,B 0,C 180,E1 -19646.657,E2 -19646.657} C_VEL
LIN {X 0,Y 234.934,Z 274.221,A -85,B 0,C 180,E1 -19650.568,E2 -19650.568} C_VEL
LIN {X 0,Y 234.961,Z 274.217,A -85,B 0,C 180,E1 -19654.633,E2 -19654.633} C_VEL
LIN {X 0,Y 234.943,Z 274.218,A -85,B 0,C 180,E1 -19658.945,E2 -19658.945} C_VEL
LIN {X 0,Y 234.878,Z 274.228,A -85,B 0,C 180,E1 -19663.488,E2 -19663.488} C_VEL
LIN {X 0,Y 234.863,Z 274.229,A -85,B 0,C 180,E1 -19666.508,E2 -19666.508} C_VEL
LIN {X 0,Y 234.892,Z 274.456,A -85,B 0,C 180,E1 -19668.834,E2 -19668.834} C_VEL
LIN {X 0,Y 235.125,Z 275.965,A -85,B 0,C 180,E1 -19671.119,E2 -19671.119} C_VEL
LIN {X 0,Y 235.178,Z 277.858,A -85,B 0,C 180,E1 -19673.791,E2 -19673.791} C_VEL
LIN {X 0,Y 234.914,Z 280.967,A -85,B 0,C 180,E1 -19677.901,E2 -19677.901} C_VEL
LIN {X 0,Y 234.87,Z 281.229,A -85,B 0,C 180,E1 -19678.234,E2 -19678.234} C_VEL
LIN {X 0,Y 235.865,Z 284.387,A -85,B 0,C 180,E1 -19678.569,E2 -19678.569} C_VEL
LIN {X 0,Y 240.292,Z 296.634,A -85,B 0,C 180,E1 -19680.052,E2 -19680.052} C_VEL
LIN {X 0,Y 243.026,Z 306.775,A -85,B 0,C 180,E1 -19681.387,E2 -19681.387} C_VEL
LIN {X 0,Y 245.074,Z 317.114,A -85,B 0,C 180,E1 -19682.893,E2 -19682.893} C_VEL
LIN {X 0,Y 246.35,Z 327.946,A -85,B 0,C 180,E1 -19684.664,E2 -19684.664} C_VEL
LIN {X 0,Y 246.197,Z 330.563,A -85,B 0,C 180,E1 -19685.099,E2 -19685.099} C_VEL
LIN {X 0,Y 243.927,Z 341.327,A -85,B 0,C 180,E1 -19686.953,E2 -19686.953} C_VEL
LIN {X 0,Y 241.95,Z 350.013,A -85,B 0,C 180,E1 -19688.829,E2 -19688.829} C_VEL
LIN {X 0,Y 239.658,Z 358.787,A -85,B 0,C 180,E1 -19691.181,E2 -19691.181} C_VEL
LIN {X 0,Y 237.562,Z 366.194,A -85,B 0,C 180,E1 -19693.677,E2 -19693.677} C_VEL
LIN {X 0,Y 235.927,Z 372.134,A -85,B 0,C 180,E1 -19696.213,E2 -19696.213} C_VEL
LIN {X 0,Y 234.656,Z 376.827,A -85,B 0,C 180,E1 -19698.774,E2 -19698.774} C_VEL
LIN {X 0,Y 233.797,Z 380.415,A -85,B 0,C 180,E1 -19701.356,E2 -19701.356} C_VEL
LIN {X 0,Y 233.18,Z 383.09,A -85,B 0,C 180,E1 -19704.053,E2 -19704.053} C_VEL
LIN {X 0,Y 232.945,Z 384.649,A -85,B 0,C 180,E1 -19706.541,E2 -19706.541} C_VEL
LIN {X 0,Y 232.834,Z 385.486,A -85,B 0,C 180,E1 -19710,E2 -19710} C_VEL
LIN {X 0,Y 232.833,Z 385.293,A -85,B 0,C 180,E1 -19711.73,E2 -19711.73} C_VEL
LIN {X 0,Y 232.944,Z 384.707,A -85,B 0,C 180,E1 -19713.46,E2 -19713.46} C_VEL
LIN {X 0,Y 233.389,Z 382.384,A -85,B 0,C 180,E1 -19716.918,E2 -19716.918} C_VEL
LIN {X 0,Y 234.071,Z 379.516,A -85,B 0,C 180,E1 -19719.505,E2 -19719.505} C_VEL
LIN {X 0,Y 235.024,Z 375.627,A -85,B 0,C 180,E1 -19722.083,E2 -19722.083} C_VEL
LIN {X 0,Y 236.412,Z 370.606,A -85,B 0,C 180,E1 -19724.637,E2 -19724.637} C_VEL
LIN {X 0,Y 238.14,Z 364.282,A -85,B 0,C 180,E1 -19727.165,E2 -19727.165} C_VEL
LIN {X 0,Y 240.351,Z 356.364,A -85,B 0,C 180,E1 -19729.65,E2 -19729.65} C_VEL
LIN {X 0,Y 242.357,Z 348.372,A -85,B 0,C 180,E1 -19731.68,E2 -19731.68} C_VEL
LIN {X 0,Y 244.579,Z 338.447,A -85,B 0,C 180,E1 -19733.722,E2 -19733.722} C_VEL
LIN {X 0,Y 246.515,Z 328.751,A -85,B 0,C 180,E1 -19735.318,E2 -19735.318} C_VEL
LIN {X 0,Y 245.224,Z 317.871,A -85,B 0,C 180,E1 -19737.125,E2 -19737.125} C_VEL
LIN {X 0,Y 242.88,Z 306.046,A -85,B 0,C 180,E1 -19738.849,E2 -19738.849} C_VEL
LIN {X 0,Y 239.859,Z 295.259,A -85,B 0,C 180,E1 -19740.261,E2 -19740.261} C_VEL
LIN {X 0,Y 235.69,Z 284.106,A -85,B 0,C 180,E1 -19741.617,E2 -19741.617} C_VEL
LIN {X 0,Y 234.847,Z 281.226,A -85,B 0,C 180,E1 -19741.925,E2 -19741.925} C_VEL
LIN {X 0,Y 235.162,Z 277.979,A -85,B 0,C 180,E1 -19746.204,E2 -19746.204} C_VEL
LIN {X 0,Y 235.105,Z 276.003,A -85,B 0,C 180,E1 -19748.993,E2 -19748.993} C_VEL
LIN {X 0,Y 234.865,Z 274.294,A -85,B 0,C 180,E1 -19751.574,E2 -19751.574} C_VEL
